  LIN {X -5735.893,Y 2029.899,Z -132.531,A -90.03341,B 0.00000,C -180.00000} ; preinsert
  LIN {X -5735.893,Y 2029.899,Z -382.531,A -90.03341,B 0.00000,C -180.00000} ; insert
  LIN {X -5735.893,Y 2029.899,Z -382.531,A -90.03341,B 0.00000,C -180.00000} ; release
  LIN {X -5735.893,Y 2029.899,Z -82.531,A -90.03341,B 0.00000,C -180.00000} ; retreat
  ; Step 3130, bar 1650
  LIN {X -5860.893,Y 2029.899,Z 855.478,A -90.03341,B 0.00000,C -180.00000} ; outside
  LIN {X -5860.893,Y 2029.899,Z -132.531,A -90.03341,B 0.00000,C -180.00000} ; preinsert
  LIN {X -5860.893,Y 2029.899,Z -382.531,A -90.03341,B 0.00000,C -180.00000} ; insert
  LIN {X -5860.893,Y 2029.899,Z -382.531,A -90.03341,B 0.00000,C -180.00000} ; release
  LIN {X -5860.893,Y 2029.899,Z -82.531,A -90.03341,B 0.00000,C -180.00000} ; retreat
  ; Step 3131, bar 1652
  LIN {X -6110.893,Y 2029.899,Z 855.478,A -90.03341,B 0.00000,C -180.00000} ; outside
  LIN {X -6110.893,Y 2029.899,Z -132.531,A -90.03341,B 0.00000,C -180.00000} ; preinsert
  LIN {X -6110.893,Y 2029.899,Z -382.531,A -90.03341,B 0.00000,C -180.00000} ; insert
  LIN {X -6110.893,Y 2029.899,Z -382.531,A -90.03341,B 0.00000,C -180.00000} ; release
  LIN {X -6110.893,Y 2029.899,Z -82.531,A -90.03341,B 0.00000,C -180.00000} ; retreat
  ; Step 3132, bar 1654
  LIN {X -6235.893,Y 2029.899,Z 855.478,A -90.03341,B 0.00000,C -180.00000} ; outside
  LIN {X -6235.893,Y 2029.899,Z -132.531,A -90.03341,B 0.00000,C -180.00000} ; preinsert
  LIN {X -6235.893,Y 2029.899,Z -382.531,A -90.03341,B 0.00000,C -180.00000} ; insert
  LIN {X -6235.893,Y 2029.899,Z -382.531,A -90.03341,B 0.00000,C -180.00000} ; release
  LIN {X -6235.893,Y 2029.899,Z -82.531,A -90.03341,B 0.00000,C -180.00000} ; retreat
  ; Step 3133, bar 1656
  LIN {X -6360.893,Y 2029.899,Z 855.478,A -90.03341,B 0.00000,C -180.00000} ; outside
  LIN {X -6360.893,Y 2029.899,Z -132.531,A -90.03341,B 0.00000,C -180.00000} ; preinsert
  LIN {X -6360.893,Y 2029.899,Z -382.531,A -90.03341,B 0.00000,C -180.00000} ; insert
  LIN {X -6360.893,Y 2029.899,Z -382.531,A -90.03341,B 0.00000,C -180.00000} ; release
  LIN {X -6360.893,Y 2029.899,Z -82.531,A -90.03341,B 0.00000,C -180.00000} ; retreat
  ; Step 3134, bar 1658
  LIN {X -6485.893,Y 2029.899,Z 855.478,A -90.03341,B 0.00000,C -180.00000} ; outside
  LIN {X -6485.893,Y 2029.899,Z -132.531,A -90.03341,B 0.00000,C -180.00000} ; preinsert
  LIN {X -6485.893,Y 2029.899,Z -382.531,A -90.03341,B 0.00000,C -180.00000} ; insert
  LIN {X -6485.893,Y 2029.899,Z -382.531,A -90.03341,B 0.00000,C -180.00000} ; release
  LIN {X -6485.893,Y 2029.899,Z -82.531,A -90.03341,B 0.00000,C -180.00000} ; retreat
  ; Step 3135, bar 1660
  LIN {X -6610.893,Y 2029.899,Z 855.478,A -90.03341,B 0.00000,C -180.00000} ; outside
  LIN {X -6610.893,Y 2029.899,Z -132.531,A -90.03341,B 0.00000,C -180.00000} ; preinsert
  LIN {X -6610.893,Y 2029.899,Z -382.531,A -90.03341,B 0.00000,C -180.00000} ; insert
  LIN {X -6610.893,Y 2029.899,Z -382.531,A -90.03341,B 0.00000,C -180.00000} ; release
  LIN {X -6610.893,Y 2029.899,Z -82.531,A -90.03341,B 0.00000,C -180.00000} ; retreat
  ; Step 3136, bar 1662
  LIN {X -6735.893,Y 2029.899,Z 855.478,A -90.03341,B 0.00000,C -180.00000} ; outside
  LIN {X -6735.893,Y 2029.899,Z -132.531,A -90.03341,B 0.00000,C -180.00000} ; preinsert
  LIN {X -6735.893,Y 2029.899,Z -382.531,A -90.03341,B 0.00000,C -180.00000} ; insert
  LIN {X -6735.893,Y 2029.899,Z -382.531,A -90.03341,B 0.00000,C -180.00000} ; release
  LIN {X -6735.893,Y 2029.899,Z -82.531,A -90.03341,B 0.00000,C -180.00000} ; retreat
  ; Step 3137, bar 1664
  LIN {X -6860.893,Y 2029.899,Z 855.478,A -90.03341,B 0.00000,C -180.00000} ; outside
  LIN {X -6860.893,Y 2029.899,Z -132.531,A -90.03341,B 0.00000,C -180.00000} ; preinsert
  LIN {X -6860.893,Y 2029.899,Z -382.531,A -90.03341,B 0.00000,C -180.00000} ; insert
  LIN {X -6860.893,Y 2029.899,Z -382.531,A -90.03341,B 0.00000,C -180.00000} ; release
  LIN {X -6860.893,Y 2029.899,Z -82.531,A -90.03341,B 0.00000,C -180.00000} ; retreat
  ; Step 3138, bar 1666
  LIN {X -6985.893,Y 2029.899,Z 855.478,A -90.03341,B 0.00000,C -180.00000} ; outside
  LIN {X -6985.893,Y 2029.899,Z -132.531,A -90.03341,B 0.00000,C -180.00000} ; preinsert
  LIN {X -6985.893,Y 2029.899,Z -382.531,A -90.03341,B 0.00000,C -180.00000} ; insert
  LIN {X -6985.893,Y 2029.899,Z -382.531,A -90.03341,B 0.00000,C -180.00000} ; release
  LIN {X -6985.893,Y 2029.899,Z -82.531,A -90.03341,B 0.00000,C -180.00000} ; retreat
  ; Step 3139, bar 1668
  LIN {X -7110.893,Y 2029.899,Z 855.478,A -90.03341,B 0.00000,C -180.00000} ; outside
  LIN {X -7110.893,Y 2029.899,Z -132.531,A -90.03341,B 0.00000,C -180.00000} ; preinsert
  LIN {X -7110.893,Y 2029.899,Z -382.531,A -90.03341,B 0.00000,C -180.00000} ; insert
  LIN {X -7110.893,Y 2029.899,Z -382.531,A -90.03341,B 0.00000,C -180.00000} ; release
  LIN {X -7110.893,Y 2029.899,Z -82.531,A -90.03341,B 0.00000,C -180.00000} ; retreat
  ; Step 3140, bar 1670
  LIN {X -7235.893,Y 2029.899,Z 855.478,A -90.03341,B 0.00000,C -180.00000} ; outside
  LIN {X -7235.893,Y 2029.899,Z -132.531,A -90.03341,B 0.00000,C -180.00000} ; preinsert
  LIN {X -7235.893,Y 2029.899,Z -382.531,A -90.03341,B 0.00000,C -180.00000} ; insert
  LIN {X -7235.893,Y 2029.899,Z -382.531,A -90.03341,B 0.00000,C -180.00000} ; release
  LIN {X -7235.893,Y 2029.899,Z -82.531,A -90.03341,B 0.00000,C -180.00000} ; retreat
  ; Step 3141, bar 1672
  LIN {X -7360.893,Y 2029.899,Z 855.478,A -90.03341,B 0.00000,C -180.00000} ; outside
  LIN {X -7360.893,Y 2029.899,Z -132.531,A -90.03341,B 0.00000,C -180.00000} ; preinsert
  LIN {X -7360.893,Y 2029.899,Z -382.531,A -90.03341,B 0.00000,C -180.00000} ; insert
  LIN {X -7360.893,Y 2029.899,Z -382.531,A -90.03341,B 0.00000,C -180.00000} ; release
  LIN {X -7360.893,Y 2029.899,Z -82.531,A -90.03341,B 0.00000,C -180.00000} ; retreat
  ; Step 3142, bar 1674
  LIN {X -7485.893,Y 2029.899,Z 855.478,A -90.03341,B 0.00000,C -180.00000} ; outside
  LIN {X -7485.893,Y 2029.899,Z -132.531,A -90.03341,B 0.00000,C -180.00000} ; preinsert
  LIN {X -7485.893,Y 2029.899,Z -382.531,A -90.03341,B 0.00000,C -180.00000} ; insert
  LIN {X -7485.893,Y 2029.899,Z -382.531,A -90.03341,B 0.00000,C -180.00000} ; release
  LIN {X -7485.893,Y 2029.899,Z -82.531,A -90.03341,B 0.00000,C -180.00000} ; retreat
  ; Step 3143, bar 1676
  LIN {X -7610.893,Y 2029.899,Z 855.478,A -90.03341,B 0.00000,C -180.00000} ; outside
  LIN {X -7610.893,Y 2029.899,Z -132.531,A -90.03341,B 0.00000,C -180.00000} ; preinsert
  LIN {X -7610.893,Y 2029.899,Z -382.531,A -90.03341,B 0.00000,C -180.00000} ; insert
  LIN {X -7610.893,Y 2029.899,Z -382.531,A -90.03341,B 0.00000,C -180.00000} ; release
  LIN {X -7610.893,Y 2029.899,Z -82.531,A -90.03341,B 0.00000,C -180.00000} ; retreat
  ; Step 3144, bar 1678
  LIN {X -7735.893,Y 2029.899,Z 855.478,A -90.03341,B 0.00000,C -180.00000} ; outside
  LIN {X -7735.893,Y 2029.899,Z -132.531,A -90.03341,B 0.00000,C -180.00000} ; preinsert
  LIN {X -7735.893,Y 2029.899,Z -382.531,A -90.03341,B 0.00000,C -180.00000} ; insert
  LIN {X -7735.893,Y 2029.899,Z -382.531,A -90.03341,B 0.00000,C -180.00000} ; release
  LIN {X -7735.893,Y 2029.899,Z -82.531,A -90.03341,B 0.00000,C -180.00000} ; retreat
  ; Step 3145, bar 1680
  LIN {X -7860.893,Y 2029.899,Z 855.478,A -90.03341,B 0.00000,C -180.00000} ; outside
  LIN {X -7860.893,Y 2029.899,Z -132.531,A -90.03341,B 0.00000,C -180.00000} ; preinsert
  LIN {X -7860.893,Y 2029.899,Z -382.531,A -90.03341,B 0.00000,C -180.00000} ; insert
  LIN {X -7860.893,Y 2029.899,Z -382.531,A -90.03341,B 0.00000,C -180.00000} ; release
  LIN {X -7860.893,Y 2029.899,Z -82.531,A -90.03341,B 0.00000,C -180.00000} ; retreat
  ; Step 3146, bar 1682
  LIN {X -7985.893,Y 2029.899,Z 855.478,A -90.03341,B 0.00000,C -180.00000} ; outside
  LIN {X -7985.893,Y 2029.899,Z -132.531,A -90.03341,B 0.00000,C -180.00000} ; preinsert
  LIN {X -7985.893,Y 2029.899,Z -382.531,A -90.03341,B 0.00000,C -180.00000} ; insert
  LIN {X -7985.893,Y 2029.899,Z -382.531,A -90.03341,B 0.00000,C -180.00000} ; release
  LIN {X -7985.893,Y 2029.899,Z -82.531,A -90.03341,B 0.00000,C -180.00000} ; retreat
  ; Step 3147, bar 1684
  LIN {X -8110.893,Y 2029.899,Z 855.478,A -90.03341,B 0.00000,C -180.00000} ; outside
  LIN {X -8110.893,Y 2029.899,Z -132.531,A -90.03341,B 0.00000,C -180.00000} ; preinsert
  LIN {X -8110.893,Y 2029.899,Z -382.531,A -90.03341,B 0.00000,C -180.00000} ; insert
  LIN {X -8110.893,Y 2029.899,Z -382.531,A -90.03341,B 0.00000,C -180.00000} ; release
  LIN {X -8110.893,Y 2029.899,Z -82.531,A -90.03341,B 0.00000,C -180.00000} ; retreat
  ; Step 3148, bar 1686
  LIN {X -8235.893,Y 2029.899,Z 855.478,A -90.03341,B 0.00000,C 180.00000} ; outside
  LIN {X -8235.893,Y 2029.899,Z -132.531,A -90.03341,B 0.00000,C 180.00000} ; preinsert
  LIN {X -8235.893,Y 2029.899,Z -382.531,A -90.03341,B 0.00000,C 180.00000} ; insert
  LIN {X -8235.893,Y 2029.899,Z -382.531,A -90.03341,B 0.00000,C 180.00000} ; release
  LIN {X -8235.893,Y 2029.899,Z -82.531,A -90.03341,B 0.00000,C 180.00000} ; retreat
  ; Step 3149, bar 1688
  LIN {X -8360.893,Y 2029.899,Z 855.478,A -90.03341,B 0.00000,C 180.00000} ; outside
  LIN {X -8360.893,Y 2029.899,Z -132.531,A -90.03341,B 0.00000,C 180.00000} ; preinsert
  LIN {X -8360.893,Y 2029.899,Z -382.531,A -90.03341,B 0.00000,C 180.00000} ; insert
  LIN {X -8360.893,Y 2029.899,Z -382.531,A -90.03341,B 0.00000,C 180.00000} ; release
  LIN {X -8360.893,Y 2029.899,Z -82.531,A -90.03341,B 0.00000,C 180.00000} ; retreat
  ; Step 3150, bar 1690
  LIN {X -8485.893,Y 2029.899,Z 855.478,A -90.03341,B 0.00000,C 180.00000} ; outside
  LIN {X -8485.893,Y 2029.899,Z -132.531,A -90.03341,B 0.00000,C 180.00000} ; preinsert
  LIN {X -8485.893,Y 2029.899,Z -382.531,A -90.03341,B 0.00000,C 180.00000} ; insert
  LIN {X -8485.893,Y 2029.899,Z -382.531,A -90.03341,B 0.00000,C 180.00000} ; release
  LIN {X -8485.893,Y 2029.899,Z -82.531,A -90.03341,B 0.00000,C 180.00000} ; retreat
  ; Step 3151, bar 1692
  LIN {X -8610.893,Y 2029.899,Z 855.478,A -90.03341,B 0.00000,C 180.00000} ; outside
  LIN {X -8610.893,Y 2029.899,Z -132.531,A -90.03341,B 0.00000,C 180.00000} ; preinsert
  LIN {X -8610.893,Y 2029.899,Z -382.531,A -90.03341,B 0.00000,C 180.00000} ; insert
  LIN {X -8610.893,Y 2029.899,Z -382.531,A -90.03341,B 0.00000,C 180.00000} ; release
  LIN {X -8610.893,Y 2029.899,Z -82.531,A -90.03341,B 0.00000,C 180.00000} ; retreat
  ; Step 3152, bar 1694
  LIN {X -8735.893,Y 2029.899,Z 855.478,A -90.03341,B 0.00000,C 180.00000} ; outside
  LIN {X -8735.893,Y 2029.899,Z -132.531,A -90.03341,B 0.00000,C 180.00000} ; preinsert
  LIN {X -8735.893,Y 2029.899,Z -382.531,A -90.03341,B 0.00000,C 180.00000} ; insert
  LIN {X -8735.893,Y 2029.899,Z -382.531,A -90.03341,B 0.00000,C 180.00000} ; release
  LIN {X -8735.893,Y 2029.899,Z -82.531,A -90.03341,B 0.00000,C 180.00000} ; retreat
  ; Step 3153, bar 1696
  LIN {X -8860.893,Y 2029.899,Z 855.478,A -90.03341,B 0.00000,C 180.00000} ; outside
  LIN {X -8860.893,Y 2029.899,Z -132.531,A -90.03341,B 0.00000,C 180.00000} ; preinsert
  LIN {X -8860.893,Y 2029.899,Z -382.531,A -90.03341,B 0.00000,C 180.00000} ; insert
  LIN {X -8860.893,Y 2029.899,Z -382.531,A -90.03341,B 0.00000,C 180.00000} ; release
  LIN {X -8860.893,Y 2029.899,Z -82.531,A -90.03341,B 0.00000,C 180.00000} ; retreat
  ; Step 3154, bar 1698
  LIN {X -8985.893,Y 2029.899,Z 855.478,A -90.03341,B 0.00000,C 180.00000} ; outside
  LIN {X -8985.893,Y 2029.899,Z -132.531,A -90.03341,B 0.00000,C 180.00000} ; preinsert
  LIN {X -8985.893,Y 2029.899,Z -382.531,A -90.03341,B 0.00000,C 180.00000} ; insert
  LIN {X -8985.893,Y 2029.899,Z -382.531,A -90.03341,B 0.00000,C 180.00000} ; release
  LIN {X -8985.893,Y 2029.899,Z -82.531,A -90.03341,B 0.00000,C 180.00000} ; retreat
  ; Step 3155, bar 1700
  LIN {X -9110.893,Y 2029.899,Z 855.478,A -90.03341,B 0.00000,C 180.00000} ; outside
  LIN {X -9110.893,Y 2029.899,Z -132.531,A -90.03341,B 0.00000,C 180.00000} ; preinsert
  LIN {X -9110.893,Y 2029.899,Z -382.531,A -90.03341,B 0.00000,C 180.00000} ; insert
  LIN {X -9110.893,Y 2029.899,Z -382.531,A -90.03341,B 0.00000,C 180.00000} ; release
  LIN {X -9110.893,Y 2029.899,Z -82.531,A -90.03341,B 0.00000,C 180.00000} ; retreat
  ; Step 3156, bar 1702
  LIN {X -9235.893,Y 2029.899,Z 855.478,A -90.03341,B 0.00000,C 180.00000} ; outside
  LIN {X -9235.893,Y 2029.899,Z -132.531,A -90.03341,B 0.00000,C 180.00000} ; preinsert
  LIN {X -9235.893,Y 2029.899,Z -382.531,A -90.03341,B 0.00000,C 180.00000} ; insert
  LIN {X -9235.893,Y 2029.899,Z -382.531,A -90.03341,B 0.00000,C 180.00000} ; release
  LIN {X -9235.893,Y 2029.899,Z -82.531,A -90.03341,B 0.00000,C 180.00000} ; retreat
  ; Step 3157, bar 1704
  LIN {X -9360.893,Y 2029.899,Z 855.478,A -90.03341,B 0.00000,C 180.00000} ; outside
  LIN {X -9360.893,Y 2029.899,Z -132.531,A -90.03341,B 0.00000,C 180.00000} ; preinsert
  LIN {X -9360.893,Y 2029.899,Z -382.531,A -90.03341,B 0.00000,C 180.00000} ; insert
  LIN {X -9360.893,Y 2029.899,Z -382.531,A -90.03341,B 0.00000,C 180.00000} ; release
  LIN {X -9360.893,Y 2029.899,Z -82.531,A -90.03341,B 0.00000,C 180.00000} ; retreat
  ; Step 3158, bar 1706
  LIN {X -9485.893,Y 2029.899,Z 855.478,A -90.03341,B 0.00000,C 180.00000} ; outside
  LIN {X -9485.893,Y 2029.899,Z -132.531,A -90.03341,B 0.00000,C 180.00000} ; preinsert
  LIN {X -9485.893,Y 2029.899,Z -382.531,A -90.03341,B 0.00000,C 180.00000} ; insert
  LIN {X -9485.893,Y 2029.899,Z -382.531,A -90.03341,B 0.00000,C 180.00000} ; release
  LIN {X -9485.893,Y 2029.899,Z -82.531,A -90.03341,B 0.00000,C 180.00000} ; retreat
  ; Step 3159, bar 1708
  LIN {X -9610.893,Y 2029.899,Z 855.478,A -90.03341,B 0.00000,C 180.00000} ; outside
  LIN {X -9610.893,Y 2029.899,Z -132.531,A -90.03341,B 0.00000,C 180.00000} ; preinsert
  LIN {X -9610.893,Y 2029.899,Z -382.531,A -90.03341,B 0.00000,C 180.00000} ; insert
  LIN {X -9610.893,Y 2029.899,Z -382.531,A -90.03341,B 0.00000,C 180.00000} ; release
  LIN {X -9610.893,Y 2029.899,Z -82.531,A -90.03341,B 0.00000,C 180.00000} ; retreat
  ; Step 3160, bar 1710
  LIN {X -9735.893,Y 2029.899,Z 855.478,A -90.03341,B 0.00000,C 180.00000} ; outside
  LIN {X -9735.893,Y 2029.899,Z -132.531,A -90.03341,B 0.00000,C 180.00000} ; preinsert
  LIN {X -9735.893,Y 2029.899,Z -382.531,A -90.03341,B 0.00000,C 180.00000} ; insert
  LIN {X -9735.893,Y 2029.899,Z -382.531,A -90.03341,B 0.00000,C 180.00000} ; release
  LIN {X -9735.893,Y 2029.899,Z -82.531,A -90.03341,B 0.00000,C 180.00000} ; retreat
  ; Step 3161, bar 1712
  LIN {X -9860.893,Y 2029.899,Z 855.478,A -90.03341,B 0.00000,C 180.00000} ; outside
  LIN {X -9860.893,Y 2029.899,Z -132.531,A -90.03341,B 0.00000,C 180.00000} ; preinsert
  LIN {X -9860.893,Y 2029.899,Z -382.531,A -90.03341,B 0.00000,C 180.00000} ; insert
  LIN {X -9860.893,Y 2029.899,Z -382.531,A -90.03341,B 0.00000,C 180.00000} ; release
  LIN {X -9860.893,Y 2029.899,Z -82.531,A -90.03341,B 0.00000,C 180.00000} ; retreat
  ; Step 3162, bar 1714
  LIN {X -10110.893,Y 2029.899,Z 855.478,A -90.03341,B 0.00000,C 180.00000} ; outside
  LIN {X -10110.893,Y 2029.899,Z -132.531,A -90.03341,B 0.00000,C 180.00000} ; preinsert
  LIN {X -10110.893,Y 2029.899,Z -382.531,A -90.03341,B 0.00000,C 180.00000} ; insert
  LIN {X -10110.893,Y 2029.899,Z -382.531,A -90.03341,B 0.00000,C 180.00000} ; release
  LIN {X -10110.893,Y 2029.899,Z -82.531,A -90.03341,B 0.00000,C 180.00000} ; retreat
  ; Step 3163, bar 1716
  LIN {X -10235.893,Y 2029.899,Z 855.478,A -90.03341,B 0.00000,C 180.00000} ; outside
  LIN {X -10235.893,Y 2029.899,Z -132.531,A -90.03341,B 0.00000,C 180.00000} ; preinsert
  LIN {X -10235.893,Y 2029.899,Z -382.531,A -90.03341,B 0.00000,C 180.00000} ; insert
  LIN {X -10235.893,Y 2029.899,Z -382.531,A -90.03341,B 0.00000,C 180.00000} ; release
  LIN {X -10235.893,Y 2029.899,Z -82.531,A -90.03341,B 0.00000,C 180.00000} ; retreat
  ; Step 3164, bar 1718
  LIN {X -10360.893,Y 2029.899,Z 855.478,A -90.03341,B 0.00000,C 180.00000} ; outside
  LIN {X -10360.893,Y 2029.899,Z -132.531,A -90.03341,B 0.00000,C 180.00000} ; preinsert
  LIN {X -10360.893,Y 2029.899,Z -382.531,A -90.03341,B 0.00000,C 180.00000} ; insert
  LIN {X -10360.893,Y 2029.899,Z -382.531,A -90.03341,B 0.00000,C 180.00000} ; release
  LIN {X -10360.893,Y 2029.899,Z -82.531,A -90.03341,B 0.00000,C 180.00000} ; retreat
  ; Step 3165, bar 1720
  LIN {X -10485.893,Y 2029.899,Z 855.478,A -90.03341,B 0.00000,C 180.00000} ; outside
  LIN {X -10485.893,Y 2029.899,Z -132.531,A -90.03341,B 0.00000,C 180.00000} ; preinsert
  LIN {X -10485.893,Y 2029.899,Z -382.531,A -90.03341,B 0.00000,C 180.00000} ; insert
  LIN {X -10485.893,Y 2029.899,Z -382.531,A -90.03341,B 0.00000,C 180.00000} ; release
  LIN {X -10485.893,Y 2029.899,Z -82.531,A -90.03341,B 0.00000,C 180.00000} ; retreat
  ; Step 3166, bar 1722
  LIN {X -10610.893,Y 2029.899,Z 855.478,A -90.03341,B 0.00000,C 180.00000} ; outside
  LIN {X -10610.893,Y 2029.899,Z -132.531,A -90.03341,B 0.00000,C 180.00000} ; preinsert
  LIN {X -10610.893,Y 2029.899,Z -382.531,A -90.03341,B 0.00000,C 180.00000} ; insert
  LIN {X -10610.893,Y 2029.899,Z -382.531,A -90.03341,B 0.00000,C 180.00000} ; release
  LIN {X -10610.893,Y 2029.899,Z -82.531,A -90.03341,B 0.00000,C 180.00000} ; retreat
  ; Step 3167, bar 1724
  LIN {X -10735.893,Y 2029.899,Z 855.478,A -90.03341,B 0.00000,C 180.00000} ; outside
  LIN {X -10735.893,Y 2029.899,Z -132.531,A -90.03341,B 0.00000,C 180.00000} ; preinsert
  LIN {X -10735.893,Y 2029.899,Z -382.531,A -90.03341,B 0.00000,C 180.00000} ; insert
  LIN {X -10735.893,Y 2029.899,Z -382.531,A -90.03341,B 0.00000,C 180.00000} ; release
  LIN {X -10735.893,Y 2029.899,Z -82.531,A -90.03341,B 0.00000,C 180.00000} ; retreat
  ; Step 3168, bar 1726
  LIN {X -10860.893,Y 2029.899,Z 855.478,A -90.03341,B 0.00000,C 180.00000} ; outside
  LIN {X -10860.893,Y 2029.899,Z -132.531,A -90.03341,B 0.00000,C 180.00000} ; preinsert
  LIN {X -10860.893,Y 2029.899,Z -382.531,A -90.03341,B 0.00000,C 180.00000} ; insert
  LIN {X -10860.893,Y 2029.899,Z -382.531,A -90.03341,B 0.00000,C 180.00000} ; release
  LIN {X -10860.893,Y 2029.899,Z -82.531,A -90.03341,B 0.00000,C 180.00000} ; retreat
  ; Step 3169, bar 1728
  LIN {X -10985.893,Y 2029.899,Z 855.478,A -90.03341,B 0.00000,C 180.00000} ; outside
  LIN {X -10985.893,Y 2029.899,Z -132.531,A -90.03341,B 0.00000,C 180.00000} ; preinsert
  LIN {X -10985.893,Y 2029.899,Z -382.531,A -90.03341,B 0.00000,C 180.00000} ; insert
  LIN {X -10985.893,Y 2029.899,Z -382.531,A -90.03341,B 0.00000,C 180.00000} ; release
  LIN {X -10985.893,Y 2029.899,Z -82.531,A -90.03341,B 0.00000,C 180.00000} ; retreat
  ; Step 3170, bar 1730
  LIN {X -11110.893,Y 2029.899,Z 855.478,A -90.03341,B 0.00000,C 180.00000} ; outside
  LIN {X -11110.893,Y 2029.899,Z -132.531,A -90.03341,B 0.00000,C 180.00000} ; preinsert
  LIN {X -11110.893,Y 2029.899,Z -382.531,A -90.03341,B 0.00000,C 180.00000} ; insert
  LIN {X -11110.893,Y 2029.899,Z -382.531,A -90.03341,B 0.00000,C 180.00000} ; release
  LIN {X -11110.893,Y 2029.899,Z -82.531,A -90.03341,B 0.00000,C 180.00000} ; retreat
  ; Step 3171, bar 1732
  LIN {X -11235.893,Y 2029.899,Z 855.478,A -90.03341,B 0.00000,C 180.00000} ; outside
  LIN {X -11235.893,Y 2029.899,Z -132.531,A -90.03341,B 0.00000,C 180.00000} ; preinsert
  LIN {X -11235.893,Y 2029.899,Z -382.531,A -90.03341,B 0.00000,C 180.00000} ; insert
  LIN {X -11235.893,Y 2029.899,Z -382.531,A -90.03341,B 0.00000,C 180.00000} ; release
  LIN {X -11235.893,Y 2029.899,Z -82.531,A -90.03341,B 0.00000,C 180.00000} ; retreat
  ; Step 3172, bar 1734
  LIN {X -11360.893,Y 2029.899,Z 855.478,A -90.03341,B 0.00000,C 180.00000} ; outside
  LIN {X -11360.893,Y 2029.899,Z -132.531,A -90.03341,B 0.00000,C 180.00000} ; preinsert
  LIN {X -11360.893,Y 2029.899,Z -382.531,A -90.03341,B 0.00000,C 180.00000} ; insert
  LIN {X -11360.893,Y 2029.899,Z -382.531,A -90.03341,B 0.00000,C 180.00000} ; release
  LIN {X -11360.893,Y 2029.899,Z -82.531,A -90.03341,B 0.00000,C 180.00000} ; retreat
  ; Step 3173, bar 1736
  LIN {X -11485.893,Y 2029.899,Z 855.478,A -90.03341,B 0.00000,C 180.00000} ; outside
  LIN {X -11485.893,Y 2029.899,Z -132.531,A -90.03341,B 0.00000,C 180.00000} ; preinsert
  LIN {X -11485.893,Y 2029.899,Z -382.531,A -90.03341,B 0.00000,C 180.00000} ; insert
  LIN {X -11485.893,Y 2029.899,Z -382.531,A -90.03341,B 0.00000,C 180.00000} ; release
  LIN {X -11485.893,Y 2029.899,Z -82.531,A -90.03341,B 0.00000,C 180.00000} ; retreat
  ; Step 3174, bar 1738
  LIN {X -11610.893,Y 2029.899,Z 855.478,A -90.03341,B 0.00000,C 180.00000} ; outside
  LIN {X -11610.893,Y 2029.899,Z -132.531,A -90.03341,B 0.00000,C 180.00000} ; preinsert
  LIN {X -11610.893,Y 2029.899,Z -382.531,A -90.03341,B 0.00000,C 180.00000} ; insert
  LIN {X -11610.893,Y 2029.899,Z -382.531,A -90.03341,B 0.00000,C 180.00000} ; release
  LIN {X -11610.893,Y 2029.899,Z -82.531,A -90.03341,B 0.00000,C 180.00000} ; retreat
  ; Step 3175, bar 1740
  LIN {X -11735.893,Y 2029.899,Z 855.478,A -90.03341,B 0.00000,C 180.00000} ; outside
  LIN {X -11735.893,Y 2029.899,Z -132.531,A -90.03341,B 0.00000,C 180.00000} ; preinsert
  LIN {X -11735.893,Y 2029.899,Z -382.531,A -90.03341,B 0.00000,C 180.00000} ; insert
  LIN {X -11735.893,Y 2029.899,Z -382.531,A -90.03341,B 0.00000,C 180.00000} ; release
  LIN {X -11735.893,Y 2029.899,Z -82.531,A -90.03341,B 0.00000,C 180.00000} ; retreat
  ; Step 3176, bar 1742
  LIN {X -11860.893,Y 2029.899,Z 855.478,A -90.03341,B 0.00000,C 180.00000} ; outside
  LIN {X -11860.893,Y 2029.899,Z -132.531,A -90.03341,B 0.00000,C 180.00000} ; preinsert
  LIN {X -11860.893,Y 2029.899,Z -382.531,A -90.03341,B 0.00000,C 180.00000} ; insert
  LIN {X -11860.893,Y 2029.899,Z -382.531,A -90.03341,B 0.00000,C 180.00000} ; release
  LIN {X -11860.893,Y 2029.899,Z -82.531,A -90.03341,B 0.00000,C 180.00000} ; retreat
  ; Step 3177, bar 1744
  LIN {X -11985.893,Y 2029.899,Z 855.478,A -90.03341,B 0.00000,C 180.00000} ; outside
  LIN {X -11985.893,Y 2029.899,Z -132.531,A -90.03341,B 0.00000,C 180.00000} ; preinsert
  LIN {X -11985.893,Y 2029.899,Z -382.531,A -90.03341,B 0.00000,C 180.00000} ; insert
  LIN {X -11985.893,Y 2029.899,Z -382.531,A -90.03341,B 0.00000,C 180.00000} ; release
  LIN {X -11985.893,Y 2029.899,Z -82.531,A -90.03341,B 0.00000,C 180.00000} ; retreat
  ; Step 3178, bar 1746
  LIN {X -12110.893,Y 2029.899,Z 855.478,A -90.03341,B 0.00000,C 180.00000} ; outside
  LIN {X -12110.893,Y 2029.899,Z -132.531,A -90.03341,B 0.00000,C 180.00000} ; preinsert
  LIN {X -12110.893,Y 2029.899,Z -382.531,A -90.03341,B 0.00000,C 180.00000} ; insert
  LIN {X -12110.893,Y 2029.899,Z -382.531,A -90.03341,B 0.00000,C 180.00000} ; release
  LIN {X -12110.893,Y 2029.899,Z -82.531,A -90.03341,B 0.00000,C 180.00000} ; retreat
  ; Step 3179, bar 1748
  LIN {X -12235.893,Y 2029.899,Z 855.478,A -90.03341,B 0.00000,C 180.00000} ; outside
  LIN {X -12235.893,Y 2029.899,Z -132.531,A -90.03341,B 0.00000,C 180.00000} ; preinsert
  LIN {X -12235.893,Y 2029.899,Z -382.531,A -90.03341,B 0.00000,C 180.00000} ; insert
  LIN {X -12235.893,Y 2029.899,Z -382.531,A -90.03341,B 0.00000,C 180.00000} ; release
  LIN {X -12235.893,Y 2029.899,Z -82.531,A -90.03341,B 0.00000,C 180.00000} ; retreat
  ; Step 3180, bar 1750
  LIN {X -12335.893,Y 2029.899,Z 855.478,A -90.03341,B 0.00000,C 180.00000} ; outside
  LIN {X -12335.893,Y 2029.899,Z -132.531,A -90.03341,B 0.00000,C 180.00000} ; preinsert
  LIN {X -12335.893,Y 2029.899,Z -382.531,A -90.03341,B 0.00000,C 180.00000} ; insert
  LIN {X -12335.893,Y 2029.899,Z -382.531,A -90.03341,B 0.00000,C 180.00000} ; release
  LIN {X -12335.893,Y 2029.899,Z -82.531,A -90.03341,B 0.00000,C 180.00000} ; retreat
  ; Step 3181, bar 1752
  LIN {X -12435.893,Y 2029.899,Z 855.478,A -90.03341,B 0.00000,C 180.00000} ; outside
  LIN {X -12435.893,Y 2029.899,Z -132.531,A -90.03341,B 0.00000,C 180.00000} ; preinsert
  LIN {X -12435.893,Y 2029.899,Z -382.531,A -90.03341,B 0.00000,C 180.00000} ; insert
  LIN {X -12435.893,Y 2029.899,Z -382.531,A -90.03341,B 0.00000,C 180.00000} ; release
  LIN {X -12435.893,Y 2029.899,Z -82.531,A -90.03341,B 0.00000,C 180.00000} ; retreat
  ; Step 3182, bar 1754
  LIN {X -12535.893,Y 2029.899,Z 855.478,A -90.03341,B 0.00000,C 180.00000} ; outside
  LIN {X -12535.893,Y 2029.899,Z -132.531,A -90.03341,B 0.00000,C 180.00000} ; preinsert
  LIN {X -12535.893,Y 2029.899,Z -382.531,A -90.03341,B 0.00000,C 180.00000} ; insert
  LIN {X -12535.893,Y 2029.899,Z -382.531,A -90.03341,B 0.00000,C 180.00000} ; release
  LIN {X -12535.893,Y 2029.899,Z -82.531,A -90.03341,B 0.00000,C 180.00000} ; retreat
  ; Step 3183, bar 1756
  LIN {X -12635.893,Y 2029.899,Z 855.478,A -90.03341,B 0.00000,C 180.00000} ; outside
  LIN {X -12635.893,Y 2029.899,Z -132.531,A -90.03341,B 0.00000,C 180.00000} ; preinsert
  LIN {X -12635.893,Y 2029.899,Z -382.531,A -90.03341,B 0.00000,C 180.00000} ; insert
  LIN {X -12635.893,Y 2029.899,Z -382.531,A -90.03341,B 0.00000,C 180.00000} ; release
  LIN {X -12635.893,Y 2029.899,Z -82.531,A -90.03341,B 0.00000,C 180.00000} ; retreat
  ; Step 3184, bar 1758
  LIN {X -12735.893,Y 2029.899,Z 855.478,A -90.03341,B 0.00000,C 180.00000} ; outside
  LIN {X -12735.893,Y 2029.899,Z -132.531,A -90.03341,B 0.00000,C 180.00000} ; preinsert
  LIN {X -12735.893,Y 2029.899,Z -382.531,A -90.03341,B 0.00000,C 180.00000} ; insert
  LIN {X -12735.893,Y 2029.899,Z -382.531,A -90.03341,B 0.00000,C 180.00000} ; release
  LIN {X -12735.893,Y 2029.899,Z -82.531,A -90.03341,B 0.00000,C 180.00000} ; retreat
  ; Step 3185, bar 1760
  LIN {X -12835.893,Y 2029.899,Z 855.478,A -90.03341,B 0.00000,C 180.00000} ; outside
  LIN {X -12835.893,Y 2029.899,Z -132.531,A -90.03341,B 0.00000,C 180.00000} ; preinsert
  LIN {X -12835.893,Y 2029.899,Z -382.531,A -90.03341,B 0.00000,C 180.00000} ; insert
  LIN {X -12835.893,Y 2029.899,Z -382.531,A -90.03341,B 0.00000,C 180.00000} ; release
  LIN {X -12835.893,Y 2029.899,Z -82.531,A -90.03341,B 0.00000,C 180.00000} ; retreat
  ; Step 3186, bar 1762
  LIN {X -12935.893,Y 2029.899,Z 855.478,A -90.03341,B 0.00000,C 180.00000} ; outside
  LIN {X -12935.893,Y 2029.899,Z -132.531,A -90.03341,B 0.00000,C 180.00000} ; preinsert
  LIN {X -12935.893,Y 2029.899,Z -382.531,A -90.03341,B 0.00000,C 180.00000} ; insert
  LIN {X -12935.893,Y 2029.899,Z -382.531,A -90.03341,B 0.00000,C 180.00000} ; release
  LIN {X -12935.893,Y 2029.899,Z -82.531,A -90.03341,B 0.00000,C 180.00000} ; retreat
  ; Step 3187, bar 1764
  LIN {X -13035.893,Y 2029.899,Z 855.478,A -90.03341,B 0.00000,C 180.00000} ; outside
  LIN {X -13035.893,Y 2029.899,Z -132.531,A -90.03341,B 0.00000,C 180.00000} ; preinsert
  LIN {X -13035.893,Y 2029.899,Z -382.531,A -90.03341,B 0.00000,C 180.00000} ; insert
  LIN {X -13035.893,Y 2029.899,Z -382.531,A -90.03341,B 0.00000,C 180.00000} ; release
  LIN {X -13035.893,Y 2029.899,Z -82.531,A -90.03341,B 0.00000,C 180.00000} ; retreat
  ; Step 3188, bar 1766
  LIN {X -13135.893,Y 2029.899,Z 855.478,A -90.03341,B 0.00000,C 180.00000} ; outside
  LIN {X -13135.893,Y 2029.899,Z -132.531,A -90.03341,B 0.00000,C 180.00000} ; preinsert
  LIN {X -13135.893,Y 2029.899,Z -382.531,A -90.03341,B 0.00000,C 180.00000} ; insert
  LIN {X -13135.893,Y 2029.899,Z -382.531,A -90.03341,B 0.00000,C 180.00000} ; release
  LIN {X -13135.893,Y 2029.899,Z -82.531,A -90.03341,B 0.00000,C 180.00000} ; retreat
  ; Step 3189, bar 1768
  LIN {X -13235.893,Y 2029.899,Z 855.478,A -90.03341,B 0.00000,C 180.00000} ; outside
  LIN {X -13235.893,Y 2029.899,Z -132.531,A -90.03341,B 0.00000,C 180.00000} ; preinsert
  LIN {X -13235.893,Y 2029.899,Z -382.531,A -90.03341,B 0.00000,C 180.00000} ; insert
  LIN {X -13235.893,Y 2029.899,Z -382.531,A -90.03341,B 0.00000,C 180.00000} ; release
  LIN {X -13235.893,Y 2029.899,Z -82.531,A -90.03341,B 0.00000,C 180.00000} ; retreat
  ; Step 3190, bar 1770
  LIN {X -13335.893,Y 2029.899,Z 855.478,A -90.03341,B 0.00000,C 180.00000} ; outside
  LIN {X -13335.893,Y 2029.899,Z -132.531,A -90.03341,B 0.00000,C 180.00000} ; preinsert
  LIN {X -13335.893,Y 2029.899,Z -382.531,A -90.03341,B 0.00000,C 180.00000} ; insert
  LIN {X -13335.893,Y 2029.899,Z -382.531,A -90.03341,B 0.00000,C 180.00000} ; release
  LIN {X -13335.893,Y 2029.899,Z -82.531,A -90.03341,B 0.00000,C 180.00000} ; retreat
  ; Step 3191, bar 1774
  LIN {X -13535.893,Y 2029.899,Z 855.478,A -90.03341,B 0.00000,C 180.00000} ; outside
  LIN {X -13535.893,Y 2029.899,Z -132.531,A -90.03341,B 0.00000,C 180.00000} ; preinsert
  LIN {X -13535.893,Y 2029.899,Z -382.531,A -90.03341,B 0.00000,C 180.00000} ; insert
  LIN {X -13535.893,Y 2029.899,Z -382.531,A -90.03341,B 0.00000,C 180.00000} ; release
  LIN {X -13535.893,Y 2029.899,Z -82.531,A -90.03341,B 0.00000,C 180.00000} ; retreat
  ; Step 3192, bar 1772
  LIN {X -13435.893,Y 2029.899,Z 855.478,A -90.03341,B 0.00000,C 180.00000} ; outside
  LIN {X -13435.893,Y 2029.899,Z -132.531,A -90.03341,B 0.00000,C 180.00000} ; preinsert
  LIN {X -13435.893,Y 2029.899,Z -382.531,A -90.03341,B 0.00000,C 180.00000} ; insert
  LIN {X -13435.893,Y 2029.899,Z -382.531,A -90.03341,B 0.00000,C 180.00000} ; release
  LIN {X -13435.893,Y 2029.899,Z -82.531,A -90.03341,B 0.00000,C 180.00000} ; retreat
  ; Step 3193, bar 1776
  LIN {X -13635.893,Y 2029.899,Z 855.478,A -90.03341,B 0.00000,C 180.00000} ; outside
  LIN {X -13635.893,Y 2029.899,Z -132.531,A -90.03341,B 0.00000,C 180.00000} ; preinsert
  LIN {X -13635.893,Y 2029.899,Z -382.531,A -90.03341,B 0.00000,C 180.00000} ; insert
  LIN {X -13635.893,Y 2029.899,Z -382.531,A -90.03341,B 0.00000,C 180.00000} ; release
  LIN {X -13635.893,Y 2029.899,Z -82.531,A -90.03341,B 0.00000,C 180.00000} ; retreat
  ; Step 3194, bar 1778
  LIN {X -13735.893,Y 2029.899,Z 855.478,A -90.03341,B 0.00000,C 180.00000} ; outside
  LIN {X -13735.893,Y 2029.899,Z -132.531,A -90.03341,B 0.00000,C 180.00000} ; preinsert
  LIN {X -13735.893,Y 2029.899,Z -382.531,A -90.03341,B 0.00000,C 180.00000} ; insert
  LIN {X -13735.893,Y 2029.899,Z -382.531,A -90.03341,B 0.00000,C 180.00000} ; release
  LIN {X -13735.893,Y 2029.899,Z -82.531,A -90.03341,B 0.00000,C 180.00000} ; retreat
  ; Step 3195, bar 1780
  LIN {X -13835.893,Y 2029.899,Z 855.478,A -90.03341,B 0.00000,C 180.00000} ; outside
  LIN {X -13835.893,Y 2029.899,Z -132.531,A -90.03341,B 0.00000,C 180.00000} ; preinsert
  LIN {X -13835.893,Y 2029.899,Z -382.531,A -90.03341,B 0.00000,C 180.00000} ; insert
  LIN {X -13835.893,Y 2029.899,Z -382.531,A -90.03341,B 0.00000,C 180.00000} ; release
  LIN {X -13835.893,Y 2029.899,Z -82.531,A -90.03341,B 0.00000,C 180.00000} ; retreat
  ; Step 3196, bar 1782
  LIN {X -14135.893,Y 2029.899,Z 855.478,A -90.03341,B 0.00000,C 180.00000} ; outside
  LIN {X -14135.893,Y 2029.899,Z -132.531,A -90.03341,B 0.00000,C 180.00000} ; preinsert
  LIN {X -14135.893,Y 2029.899,Z -382.531,A -90.03341,B 0.00000,C 180.00000} ; insert
  LIN {X -14135.893,Y 2029.899,Z -382.531,A -90.03341,B 0.00000,C 180.00000} ; release
  LIN {X -14135.893,Y 2029.899,Z -82.531,A -90.03341,B 0.00000,C 180.00000} ; retreat
  ; Step 3197, bar 1784
  LIN {X -14235.893,Y 2029.899,Z 855.478,A -90.03341,B 0.00000,C 180.00000} ; outside
  LIN {X -14235.893,Y 2029.899,Z -132.531,A -90.03341,B 0.00000,C 180.00000} ; preinsert
  LIN {X -14235.893,Y 2029.899,Z -382.531,A -90.03341,B 0.00000,C 180.00000} ; insert
  LIN {X -14235.893,Y 2029.899,Z -382.531,A -90.03341,B 0.00000,C 180.00000} ; release
  LIN {X -14235.893,Y 2029.899,Z -82.531,A -90.03341,B 0.00000,C 180.00000} ; retreat
  ; Step 3198, bar 1252
  LIN {X -14.107,Y 2029.899,Z 855.478,A -89.96659,B 0.00000,C 180.00000} ; outside
  LIN {X -14.107,Y 2029.899,Z -132.531,A -89.96659,B 0.00000,C 180.00000} ; preinsert
  LIN {X -14.107,Y 2029.899,Z -382.531,A -89.96659,B 0.00000,C 180.00000} ; insert
  LIN {X -14.107,Y 2029.899,Z -382.531,A -89.96659,B 0.00000,C 180.00000} ; release
  LIN {X -14.107,Y 2029.899,Z -82.531,A -89.96659,B 0.00000,C 180.00000} ; retreat
  ; Step 3199, bar 1254
  LIN {X 110.893,Y 2029.899,Z 855.478,A -89.96659,B 0.00000,C 180.00000} ; outside
  LIN {X 110.893,Y 2029.899,Z -132.531,A -89.96659,B 0.00000,C 180.00000} ; preinsert
  LIN {X 110.893,Y 2029.899,Z -382.531,A -89.96659,B 0.00000,C 180.00000} ; insert
  LIN {X 110.893,Y 2029.899,Z -382.531,A -89.96659,B 0.00000,C 180.00000} ; release
  LIN {X 110.893,Y 2029.899,Z -82.531,A -89.96659,B 0.00000,C 180.00000} ; retreat
  ; Step 3200, bar 1256
  LIN {X 235.893,Y 2029.899,Z 855.478,A -89.96659,B 0.00000,C 180.00000} ; outside
  LIN {X 235.893,Y 2029.899,Z -132.531,A -89.96659,B 0.00000,C 180.00000} ; preinsert
  LIN {X 235.893,Y 2029.899,Z -382.531,A -89.96659,B 0.00000,C 180.00000} ; insert
  LIN {X 235.893,Y 2029.899,Z -382.531,A -89.96659,B 0.00000,C 180.00000} ; release
  LIN {X 235.893,Y 2029.899,Z -82.531,A -89.96659,B 0.00000,C 180.00000} ; retreat
  ; Step 3201, bar 1258
  LIN {X 360.893,Y 2029.899,Z 855.478,A -89.96659,B 0.00000,C 180.00000} ; outside
  LIN {X 360.893,Y 2029.899,Z -132.531,A -89.96659,B 0.00000,C 180.00000} ; preinsert
  LIN {X 360.893,Y 2029.899,Z -382.531,A -89.96659,B 0.00000,C 180.00000} ; insert
  LIN {X 360.893,Y 2029.899,Z -382.531,A -89.96659,B 0.00000,C 180.00000} ; release
  LIN {X 360.893,Y 2029.899,Z -82.531,A -89.96659,B 0.00000,C 180.00000} ; retreat
  ; Step 3202, bar 1260
  LIN {X 485.893,Y 2029.899,Z 855.478,A -89.96659,B 0.00000,C 180.00000} ; outside
  LIN {X 485.893,Y 2029.899,Z -132.531,A -89.96659,B 0.00000,C 180.00000} ; preinsert
  LIN {X 485.893,Y 2029.899,Z -382.531,A -89.96659,B 0.00000,C 180.00000} ; insert
  LIN {X 485.893,Y 2029.899,Z -382.531,A -89.96659,B 0.00000,C 180.00000} ; release
  LIN {X 485.893,Y 2029.899,Z -82.531,A -89.96659,B 0.00000,C 180.00000} ; retreat
  ; Step 3203, bar 1262
  LIN {X 610.893,Y 2029.899,Z 855.478,A -89.96659,B 0.00000,C 180.00000} ; outside
  LIN {X 610.893,Y 2029.899,Z -132.531,A -89.96659,B 0.00000,C 180.00000} ; preinsert
  LIN {X 610.893,Y 2029.899,Z -382.531,A -89.96659,B 0.00000,C 180.00000} ; insert
  LIN {X 610.893,Y 2029.899,Z -382.531,A -89.96659,B 0.00000,C 180.00000} ; release
  LIN {X 610.893,Y 2029.899,Z -82.531,A -89.96659,B 0.00000,C 180.00000} ; retreat
  ; Step 3204, bar 1264
  LIN {X 735.893,Y 2029.899,Z 855.478,A -89.96659,B 0.00000,C 180.00000} ; outside
  LIN {X 735.893,Y 2029.899,Z -132.531,A -89.96659,B 0.00000,C 180.00000} ; preinsert
  LIN {X 735.893,Y 2029.899,Z -382.531,A -89.96659,B 0.00000,C 180.00000} ; insert
  LIN {X 735.893,Y 2029.899,Z -382.531,A -89.96659,B 0.00000,C 180.00000} ; release
  LIN {X 735.893,Y 2029.899,Z -82.531,A -89.96659,B 0.00000,C 180.00000} ; retreat
  ; Step 3205, bar 1266
  LIN {X 860.893,Y 2029.899,Z 855.478,A -89.96659,B 0.00000,C 180.00000} ; outside
  LIN {X 860.893,Y 2029.899,Z -132.531,A -89.96659,B 0.00000,C 180.00000} ; preinsert
  LIN {X 860.893,Y 2029.899,Z -382.531,A -89.96659,B 0.00000,C 180.00000} ; insert
  LIN {X 860.893,Y 2029.899,Z -382.531,A -89.96659,B 0.00000,C 180.00000} ; release
  LIN {X 860.893,Y 2029.899,Z -82.531,A -89.96659,B 0.00000,C 180.00000} ; retreat
  ; Step 3206, bar 1268
  LIN {X 985.893,Y 2029.899,Z 855.478,A -89.96659,B 0.00000,C 180.00000} ; outside
  LIN {X 985.893,Y 2029.899,Z -132.531,A -89.96659,B 0.00000,C 180.00000} ; preinsert
  LIN {X 985.893,Y 2029.899,Z -382.531,A -89.96659,B 0.00000,C 180.00000} ; insert
  LIN {X 985.893,Y 2029.899,Z -382.531,A -89.96659,B 0.00000,C 180.00000} ; release
  LIN {X 985.893,Y 2029.899,Z -82.531,A -89.96659,B 0.00000,C 180.00000} ; retreat
  ; Step 3207, bar 1270
  LIN {X 1110.893,Y 2029.899,Z 855.478,A -89.96659,B 0.00000,C 180.00000} ; outside
  LIN {X 1110.893,Y 2029.899,Z -132.531,A -89.96659,B 0.00000,C 180.00000} ; preinsert
  LIN {X 1110.893,Y 2029.899,Z -382.531,A -89.96659,B 0.00000,C 180.00000} ; insert
  LIN {X 1110.893,Y 2029.899,Z -382.531,A -89.96659,B 0.00000,C 180.00000} ; release
  LIN {X 1110.893,Y 2029.899,Z -82.531,A -89.96659,B 0.00000,C 180.00000} ; retreat
  ; Step 3208, bar 1272
  LIN {X 1235.893,Y 2029.899,Z 855.478,A -89.96659,B 0.00000,C 180.00000} ; outside
  LIN {X 1235.893,Y 2029.899,Z -132.531,A -89.96659,B 0.00000,C 180.00000} ; preinsert
  LIN {X 1235.893,Y 2029.899,Z -382.531,A -89.96659,B 0.00000,C 180.00000} ; insert
  LIN {X 1235.893,Y 2029.899,Z -382.531,A -89.96659,B 0.00000,C 180.00000} ; release
  LIN {X 1235.893,Y 2029.899,Z -82.531,A -89.96659,B 0.00000,C 180.00000} ; retreat
  ; Step 3209, bar 1274
  LIN {X 1360.893,Y 2029.899,Z 855.478,A -89.96659,B 0.00000,C 180.00000} ; outside
  LIN {X 1360.893,Y 2029.899,Z -132.531,A -89.96659,B 0.00000,C 180.00000} ; preinsert
  LIN {X 1360.893,Y 2029.899,Z -382.531,A -89.96659,B 0.00000,C 180.00000} ; insert
  LIN {X 1360.893,Y 2029.899,Z -382.531,A -89.96659,B 0.00000,C 180.00000} ; release
  LIN {X 1360.893,Y 2029.899,Z -82.531,A -89.96659,B 0.00000,C 180.00000} ; retreat
  ; Step 3210, bar 1276
  LIN {X 1485.893,Y 2029.899,Z 855.478,A -89.96659,B 0.00000,C 180.00000} ; outside
  LIN {X 1485.893,Y 2029.899,Z -132.531,A -89.96659,B 0.00000,C 180.00000} ; preinsert
  LIN {X 1485.893,Y 2029.899,Z -382.531,A -89.96659,B 0.00000,C 180.00000} ; insert
  LIN {X 1485.893,Y 2029.899,Z -382.531,A -89.96659,B 0.00000,C 180.00000} ; release
  LIN {X 1485.893,Y 2029.899,Z -82.531,A -89.96659,B 0.00000,C 180.00000} ; retreat
  ; Step 3211, bar 1278
  LIN {X 1610.893,Y 2029.899,Z 855.478,A -89.96659,B 0.00000,C 180.00000} ; outside
  LIN {X 1610.893,Y 2029.899,Z -132.531,A -89.96659,B 0.00000,C 180.00000} ; preinsert
  LIN {X 1610.893,Y 2029.899,Z -382.531,A -89.96659,B 0.00000,C 180.00000} ; insert
  LIN {X 1610.893,Y 2029.899,Z -382.531,A -89.96659,B 0.00000,C 180.00000} ; release
  LIN {X 1610.893,Y 2029.899,Z -82.531,A -89.96659,B 0.00000,C 180.00000} ; retreat
  ; Step 3212, bar 1280
  LIN {X 1735.893,Y 2029.899,Z 855.478,A -89.96659,B 0.00000,C 180.00000} ; outside
  LIN {X 1735.893,Y 2029.899,Z -132.531,A -89.96659,B 0.00000,C 180.00000} ; preinsert
  LIN {X 1735.893,Y 2029.899,Z -382.531,A -89.96659,B 0.00000,C 180.00000} ; insert
  LIN {X 1735.893,Y 2029.899,Z -382.531,A -89.96659,B 0.00000,C 180.00000} ; release
  LIN {X 1735.893,Y 2029.899,Z -82.531,A -89.96659,B 0.00000,C 180.00000} ; retreat
  ; Step 3213, bar 1282
  LIN {X 1860.893,Y 2029.899,Z 855.478,A -89.96659,B 0.00000,C 180.00000} ; outside
  LIN {X 1860.893,Y 2029.899,Z -132.531,A -89.96659,B 0.00000,C 180.00000} ; preinsert
  LIN {X 1860.893,Y 2029.899,Z -382.531,A -89.96659,B 0.00000,C 180.00000} ; insert
  LIN {X 1860.893,Y 2029.899,Z -382.531,A -89.96659,B 0.00000,C 180.00000} ; release
  LIN {X 1860.893,Y 2029.899,Z -82.531,A -89.96659,B 0.00000,C 180.00000} ; retreat
  ; Step 3214, bar 1284
  LIN {X 2110.893,Y 2029.899,Z 855.478,A -89.96659,B 0.00000,C 180.00000} ; outside
  LIN {X 2110.893,Y 2029.899,Z -132.531,A -89.96659,B 0.00000,C 180.00000} ; preinsert
  LIN {X 2110.893,Y 2029.899,Z -382.531,A -89.96659,B 0.00000,C 180.00000} ; insert
  LIN {X 2110.893,Y 2029.899,Z -382.531,A -89.96659,B 0.00000,C 180.00000} ; release
  LIN {X 2110.893,Y 2029.899,Z -82.531,A -89.96659,B 0.00000,C 180.00000} ; retreat
  ; Step 3215, bar 1286
  LIN {X 2235.893,Y 2029.899,Z 855.478,A -89.96659,B 0.00000,C 180.00000} ; outside
  LIN {X 2235.893,Y 2029.899,Z -132.531,A -89.96659,B 0.00000,C 180.00000} ; preinsert
  LIN {X 2235.893,Y 2029.899,Z -382.531,A -89.96659,B 0.00000,C 180.00000} ; insert
  LIN {X 2235.893,Y 2029.899,Z -382.531,A -89.96659,B 0.00000,C 180.00000} ; release
  LIN {X 2235.893,Y 2029.899,Z -82.531,A -89.96659,B 0.00000,C 180.00000} ; retreat
  ; Step 3216, bar 1288
  LIN {X 2360.893,Y 2029.899,Z 855.478,A -89.96659,B 0.00000,C 180.00000} ; outside
  LIN {X 2360.893,Y 2029.899,Z -132.531,A -89.96659,B 0.00000,C 180.00000} ; preinsert
  LIN {X 2360.893,Y 2029.899,Z -382.531,A -89.96659,B 0.00000,C 180.00000} ; insert
  LIN {X 2360.893,Y 2029.899,Z -382.531,A -89.96659,B 0.00000,C 180.00000} ; release
  LIN {X 2360.893,Y 2029.899,Z -82.531,A -89.96659,B 0.00000,C 180.00000} ; retreat
  ; Step 3217, bar 1290
  LIN {X 2485.893,Y 2029.899,Z 855.478,A -89.96659,B 0.00000,C 180.00000} ; outside
  LIN {X 2485.893,Y 2029.899,Z -132.531,A -89.96659,B 0.00000,C 180.00000} ; preinsert
  LIN {X 2485.893,Y 2029.899,Z -382.531,A -89.96659,B 0.00000,C 180.00000} ; insert
  LIN {X 2485.893,Y 2029.899,Z -382.531,A -89.96659,B 0.00000,C 180.00000} ; release
  LIN {X 2485.893,Y 2029.899,Z -82.531,A -89.96659,B 0.00000,C 180.00000} ; retreat
  ; Step 3218, bar 1292
  LIN {X 2610.893,Y 2029.899,Z 855.478,A -89.96659,B 0.00000,C 180.00000} ; outside
  LIN {X 2610.893,Y 2029.899,Z -132.531,A -89.96659,B 0.00000,C 180.00000} ; preinsert
  LIN {X 2610.893,Y 2029.899,Z -382.531,A -89.96659,B 0.00000,C 180.00000} ; insert
  LIN {X 2610.893,Y 2029.899,Z -382.531,A -89.96659,B 0.00000,C 180.00000} ; release
  LIN {X 2610.893,Y 2029.899,Z -82.531,A -89.96659,B 0.00000,C 180.00000} ; retreat
  ; Step 3219, bar 1294
  LIN {X 2735.893,Y 2029.899,Z 855.478,A -89.96659,B 0.00000,C 180.00000} ; outside
  LIN {X 2735.893,Y 2029.899,Z -132.531,A -89.96659,B 0.00000,C 180.00000} ; preinsert
  LIN {X 2735.893,Y 2029.899,Z -382.531,A -89.96659,B 0.00000,C 180.00000} ; insert
  LIN {X 2735.893,Y 2029.899,Z -382.531,A -89.96659,B 0.00000,C 180.00000} ; release
  LIN {X 2735.893,Y 2029.899,Z -82.531,A -89.96659,B 0.00000,C 180.00000} ; retreat
  ; Step 3220, bar 1296
  LIN {X 2860.893,Y 2029.899,Z 855.478,A -89.96659,B 0.00000,C 180.00000} ; outside
  LIN {X 2860.893,Y 2029.899,Z -132.531,A -89.96659,B 0.00000,C 180.00000} ; preinsert
  LIN {X 2860.893,Y 2029.899,Z -382.531,A -89.96659,B 0.00000,C 180.00000} ; insert
  LIN {X 2860.893,Y 2029.899,Z -382.531,A -89.96659,B 0.00000,C 180.00000} ; release
  LIN {X 2860.893,Y 2029.899,Z -82.531,A -89.96659,B 0.00000,C 180.00000} ; retreat
  ; Step 3221, bar 1298
  LIN {X 2985.893,Y 2029.899,Z 855.478,A -89.96659,B 0.00000,C 180.00000} ; outside
  LIN {X 2985.893,Y 2029.899,Z -132.531,A -89.96659,B 0.00000,C 180.00000} ; preinsert
  LIN {X 2985.893,Y 2029.899,Z -382.531,A -89.96659,B 0.00000,C 180.00000} ; insert
  LIN {X 2985.893,Y 2029.899,Z -382.531,A -89.96659,B 0.00000,C 180.00000} ; release
  LIN {X 2985.893,Y 2029.899,Z -82.531,A -89.96659,B 0.00000,C 180.00000} ; retreat
  ; Step 3222, bar 1300
  LIN {X 3110.893,Y 2029.899,Z 855.478,A -89.96659,B 0.00000,C 180.00000} ; outside
  LIN {X 3110.893,Y 2029.899,Z -132.531,A -89.96659,B 0.00000,C 180.00000} ; preinsert
  LIN {X 3110.893,Y 2029.899,Z -382.531,A -89.96659,B 0.00000,C 180.00000} ; insert
  LIN {X 3110.893,Y 2029.899,Z -382.531,A -89.96659,B 0.00000,C 180.00000} ; release
  LIN {X 3110.893,Y 2029.899,Z -82.531,A -89.96659,B 0.00000,C 180.00000} ; retreat
  ; Step 3223, bar 1302
  LIN {X 3235.893,Y 2029.899,Z 855.478,A -89.96659,B 0.00000,C 180.00000} ; outside
  LIN {X 3235.893,Y 2029.899,Z -132.531,A -89.96659,B 0.00000,C 180.00000} ; preinsert
  LIN {X 3235.893,Y 2029.899,Z -382.531,A -89.96659,B 0.00000,C 180.00000} ; insert
  LIN {X 3235.893,Y 2029.899,Z -382.531,A -89.96659,B 0.00000,C 180.00000} ; release
  LIN {X 3235.893,Y 2029.899,Z -82.531,A -89.96659,B 0.00000,C 180.00000} ; retreat
  ; Step 3224, bar 1304
  LIN {X 3360.893,Y 2029.899,Z 855.478,A -89.96659,B 0.00000,C 180.00000} ; outside
  LIN {X 3360.893,Y 2029.899,Z -132.531,A -89.96659,B 0.00000,C 180.00000} ; preinsert
  LIN {X 3360.893,Y 2029.899,Z -382.531,A -89.96659,B 0.00000,C 180.00000} ; insert
  LIN {X 3360.893,Y 2029.899,Z -382.531,A -89.96659,B 0.00000,C 180.00000} ; release
  LIN {X 3360.893,Y 2029.899,Z -82.531,A -89.96659,B 0.00000,C 180.00000} ; retreat
  ; Step 3225, bar 1306
  LIN {X 3485.893,Y 2029.899,Z 855.478,A -89.96659,B 0.00000,C 180.00000} ; outside
  LIN {X 3485.893,Y 2029.899,Z -132.531,A -89.96659,B 0.00000,C 180.00000} ; preinsert
  LIN {X 3485.893,Y 2029.899,Z -382.531,A -89.96659,B 0.00000,C 180.00000} ; insert
  LIN {X 3485.893,Y 2029.899,Z -382.531,A -89.96659,B 0.00000,C 180.00000} ; release
  LIN {X 3485.893,Y 2029.899,Z -82.531,A -89.96659,B 0.00000,C 180.00000} ; retreat
  ; Step 3226, bar 1308
  LIN {X 3610.893,Y 2029.899,Z 855.478,A -89.96659,B 0.00000,C 180.00000} ; outside
  LIN {X 3610.893,Y 2029.899,Z -132.531,A -89.96659,B 0.00000,C 180.00000} ; preinsert
  LIN {X 3610.893,Y 2029.899,Z -382.531,A -89.96659,B 0.00000,C 180.00000} ; insert
  LIN {X 3610.893,Y 2029.899,Z -382.531,A -89.96659,B 0.00000,C 180.00000} ; release
  LIN {X 3610.893,Y 2029.899,Z -82.531,A -89.96659,B 0.00000,C 180.00000} ; retreat
  ; Step 3227, bar 1310
  LIN {X 3735.893,Y 2029.899,Z 855.478,A -89.96659,B 0.00000,C 180.00000} ; outside
  LIN {X 3735.893,Y 2029.899,Z -132.531,A -89.96659,B 0.00000,C 180.00000} ; preinsert
  LIN {X 3735.893,Y 2029.899,Z -382.531,A -89.96659,B 0.00000,C 180.00000} ; insert
  LIN {X 3735.893,Y 2029.899,Z -382.531,A -89.96659,B 0.00000,C 180.00000} ; release
  LIN {X 3735.893,Y 2029.899,Z -82.531,A -89.96659,B 0.00000,C 180.00000} ; retreat
  ; Step 3228, bar 1312
  LIN {X 3860.893,Y 2029.899,Z 855.478,A -89.96659,B 0.00000,C 180.00000} ; outside
  LIN {X 3860.893,Y 2029.899,Z -132.531,A -89.96659,B 0.00000,C 180.00000} ; preinsert
  LIN {X 3860.893,Y 2029.899,Z -382.531,A -89.96659,B 0.00000,C 180.00000} ; insert
  LIN {X 3860.893,Y 2029.899,Z -382.531,A -89.96659,B 0.00000,C 180.00000} ; release
  LIN {X 3860.893,Y 2029.899,Z -82.531,A -89.96659,B 0.00000,C 180.00000} ; retreat
  ; Step 3229, bar 1314
  LIN {X 3985.893,Y 2029.899,Z 855.478,A -89.96659,B 0.00000,C 180.00000} ; outside
  LIN {X 3985.893,Y 2029.899,Z -132.531,A -89.96659,B 0.00000,C 180.00000} ; preinsert
  LIN {X 3985.893,Y 2029.899,Z -382.531,A -89.96659,B 0.00000,C 180.00000} ; insert
  LIN {X 3985.893,Y 2029.899,Z -382.531,A -89.96659,B 0.00000,C 180.00000} ; release
  LIN {X 3985.893,Y 2029.899,Z -82.531,A -89.96659,B 0.00000,C 180.00000} ; retreat
  ; Step 3230, bar 1316
  LIN {X 4110.893,Y 2029.899,Z 855.478,A -89.96659,B 0.00000,C 180.00000} ; outside
  LIN {X 4110.893,Y 2029.899,Z -132.531,A -89.96659,B 0.00000,C 180.00000} ; preinsert
  LIN {X 4110.893,Y 2029.899,Z -382.531,A -89.96659,B 0.00000,C 180.00000} ; insert
  LIN {X 4110.893,Y 2029.899,Z -382.531,A -89.96659,B 0.00000,C 180.00000} ; release
  LIN {X 4110.893,Y 2029.899,Z -82.531,A -89.96659,B 0.00000,C 180.00000} ; retreat
  ; Step 3231, bar 1318
  LIN {X 4235.893,Y 2029.899,Z 855.478,A -89.96659,B 0.00000,C 180.00000} ; outside
  LIN {X 4235.893,Y 2029.899,Z -132.531,A -89.96659,B 0.00000,C 180.00000} ; preinsert
  LIN {X 4235.893,Y 2029.899,Z -382.531,A -89.96659,B 0.00000,C 180.00000} ; insert
  LIN {X 4235.893,Y 2029.899,Z -382.531,A -89.96659,B 0.00000,C 180.00000} ; release
  LIN {X 4235.893,Y 2029.899,Z -82.531,A -89.96659,B 0.00000,C 180.00000} ; retreat
  ; Step 3232, bar 1320
  LIN {X 4360.893,Y 2029.899,Z 855.478,A -89.96659,B 0.00000,C 180.00000} ; outside
  LIN {X 4360.893,Y 2029.899,Z -132.531,A -89.96659,B 0.00000,C 180.00000} ; preinsert
  LIN {X 4360.893,Y 2029.899,Z -382.531,A -89.96659,B 0.00000,C 180.00000} ; insert
  LIN {X 4360.893,Y 2029.899,Z -382.531,A -89.96659,B 0.00000,C 180.00000} ; release
  LIN {X 4360.893,Y 2029.899,Z -82.531,A -89.96659,B 0.00000,C 180.00000} ; retreat
  ; Step 3233, bar 1322
  LIN {X 4485.893,Y 2029.899,Z 855.478,A -89.96659,B 0.00000,C 180.00000} ; outside
  LIN {X 4485.893,Y 2029.899,Z -132.531,A -89.96659,B 0.00000,C 180.00000} ; preinsert
  LIN {X 4485.893,Y 2029.899,Z -382.531,A -89.96659,B 0.00000,C 180.00000} ; insert
  LIN {X 4485.893,Y 2029.899,Z -382.531,A -89.96659,B 0.00000,C 180.00000} ; release
  LIN {X 4485.893,Y 2029.899,Z -82.531,A -89.96659,B 0.00000,C 180.00000} ; retreat
  ; Step 3234, bar 1324
  LIN {X 4610.893,Y 2029.899,Z 855.478,A -89.96659,B 0.00000,C 180.00000} ; outside
  LIN {X 4610.893,Y 2029.899,Z -132.531,A -89.96659,B 0.00000,C 180.00000} ; preinsert
  LIN {X 4610.893,Y 2029.899,Z -382.531,A -89.96659,B 0.00000,C 180.00000} ; insert
  LIN {X 4610.893,Y 2029.899,Z -382.531,A -89.96659,B 0.00000,C 180.00000} ; release
  LIN {X 4610.893,Y 2029.899,Z -82.531,A -89.96659,B 0.00000,C 180.00000} ; retreat
  ; Step 3235, bar 1326
  LIN {X 4735.893,Y 2029.899,Z 855.478,A -89.96659,B 0.00000,C 180.00000} ; outside
  LIN {X 4735.893,Y 2029.899,Z -132.531,A -89.96659,B 0.00000,C 180.00000} ; preinsert
  LIN {X 4735.893,Y 2029.899,Z -382.531,A -89.96659,B 0.00000,C 180.00000} ; insert
  LIN {X 4735.893,Y 2029.899,Z -382.531,A -89.96659,B 0.00000,C 180.00000} ; release
  LIN {X 4735.893,Y 2029.899,Z -82.531,A -89.96659,B 0.00000,C 180.00000} ; retreat
  ; Step 3236, bar 1328
  LIN {X 4860.893,Y 2029.899,Z 855.478,A -89.96659,B 0.00000,C 180.00000} ; outside
  LIN {X 4860.893,Y 2029.899,Z -132.531,A -89.96659,B 0.00000,C 180.00000} ; preinsert
  LIN {X 4860.893,Y 2029.899,Z -382.531,A -89.96659,B 0.00000,C 180.00000} ; insert
  LIN {X 4860.893,Y 2029.899,Z -382.531,A -89.96659,B 0.00000,C 180.00000} ; release
  LIN {X 4860.893,Y 2029.899,Z -82.531,A -89.96659,B 0.00000,C 180.00000} ; retreat
  ; Step 3237, bar 1330
  LIN {X 4985.893,Y 2029.899,Z 855.478,A -89.96659,B 0.00000,C 180.00000} ; outside
  LIN {X 4985.893,Y 2029.899,Z -132.531,A -89.96659,B 0.00000,C 180.00000} ; preinsert
  LIN {X 4985.893,Y 2029.899,Z -382.531,A -89.96659,B 0.00000,C 180.00000} ; insert
  LIN {X 4985.893,Y 2029.899,Z -382.531,A -89.96659,B 0.00000,C 180.00000} ; release
  LIN {X 4985.893,Y 2029.899,Z -82.531,A -89.96659,B 0.00000,C 180.00000} ; retreat
  ; Step 3238, bar 1332
  LIN {X 5110.893,Y 2029.899,Z 855.478,A -89.96659,B 0.00000,C 180.00000} ; outside
  LIN {X 5110.893,Y 2029.899,Z -132.531,A -89.96659,B 0.00000,C 180.00000} ; preinsert
  LIN {X 5110.893,Y 2029.899,Z -382.531,A -89.96659,B 0.00000,C 180.00000} ; insert
  LIN {X 5110.893,Y 2029.899,Z -382.531,A -89.96659,B 0.00000,C 180.00000} ; release
  LIN {X 5110.893,Y 2029.899,Z -82.531,A -89.96659,B 0.00000,C 180.00000} ; retreat
  ; Step 3239, bar 1334
  LIN {X 5235.893,Y 2029.899,Z 855.478,A -89.96659,B 0.00000,C 180.00000} ; outside
  LIN {X 5235.893,Y 2029.899,Z -132.531,A -89.96659,B 0.00000,C 180.00000} ; preinsert
  LIN {X 5235.893,Y 2029.899,Z -382.531,A -89.96659,B 0.00000,C 180.00000} ; insert
  LIN {X 5235.893,Y 2029.899,Z -382.531,A -89.96659,B 0.00000,C 180.00000} ; release
  LIN {X 5235.893,Y 2029.899,Z -82.531,A -89.96659,B 0.00000,C 180.00000} ; retreat
  ; Step 3240, bar 1336
  LIN {X 5360.893,Y 2029.899,Z 855.478,A -89.96659,B 0.00000,C 180.00000} ; outside
  LIN {X 5360.893,Y 2029.899,Z -132.531,A -89.96659,B 0.00000,C 180.00000} ; preinsert
  LIN {X 5360.893,Y 2029.899,Z -382.531,A -89.96659,B 0.00000,C 180.00000} ; insert
  LIN {X 5360.893,Y 2029.899,Z -382.531,A -89.96659,B 0.00000,C 180.00000} ; release
  LIN {X 5360.893,Y 2029.899,Z -82.531,A -89.96659,B 0.00000,C 180.00000} ; retreat
  ; Step 3241, bar 1338
  LIN {X 5485.893,Y 2029.899,Z 855.478,A -89.96659,B 0.00000,C 180.00000} ; outside
  LIN {X 5485.893,Y 2029.899,Z -132.531,A -89.96659,B 0.00000,C 180.00000} ; preinsert
  LIN {X 5485.893,Y 2029.899,Z -382.531,A -89.96659,B 0.00000,C 180.00000} ; insert
  LIN {X 5485.893,Y 2029.899,Z -382.531,A -89.96659,B 0.00000,C 180.00000} ; release
  LIN {X 5485.893,Y 2029.899,Z -82.531,A -89.96659,B 0.00000,C 180.00000} ; retreat
  ; Step 3242, bar 1340
  LIN {X 5610.893,Y 2029.899,Z 855.478,A -89.96659,B 0.00000,C 180.00000} ; outside
  LIN {X 5610.893,Y 2029.899,Z -132.531,A -89.96659,B 0.00000,C 180.00000} ; preinsert
  LIN {X 5610.893,Y 2029.899,Z -382.531,A -89.96659,B 0.00000,C 180.00000} ; insert
  LIN {X 5610.893,Y 2029.899,Z -382.531,A -89.96659,B 0.00000,C 180.00000} ; release
  LIN {X 5610.893,Y 2029.899,Z -82.531,A -89.96659,B 0.00000,C 180.00000} ; retreat
  ; Step 3243, bar 1342
  LIN {X 5735.893,Y 2029.899,Z 855.478,A -89.96659,B 0.00000,C 180.00000} ; outside
  LIN {X 5735.893,Y 2029.899,Z -132.531,A -89.96659,B 0.00000,C 180.00000} ; preinsert
  LIN {X 5735.893,Y 2029.899,Z -382.531,A -89.96659,B 0.00000,C 180.00000} ; insert
  LIN {X 5735.893,Y 2029.899,Z -382.531,A -89.96659,B 0.00000,C 180.00000} ; release
  LIN {X 5735.893,Y 2029.899,Z -82.531,A -89.96659,B 0.00000,C 180.00000} ; retreat
  ; Step 3244, bar 1344
  LIN {X 5860.893,Y 2029.899,Z 855.478,A -89.96659,B 0.00000,C 180.00000} ; outside
  LIN {X 5860.893,Y 2029.899,Z -132.531,A -89.96659,B 0.00000,C 180.00000} ; preinsert
  LIN {X 5860.893,Y 2029.899,Z -382.531,A -89.96659,B 0.00000,C 180.00000} ; insert
  LIN {X 5860.893,Y 2029.899,Z -382.531,A -89.96659,B 0.00000,C 180.00000} ; release
  LIN {X 5860.893,Y 2029.899,Z -82.531,A -89.96659,B 0.00000,C 180.00000} ; retreat
  ; Step 3245, bar 1346
  LIN {X 6110.893,Y 2029.899,Z 855.478,A -89.96659,B 0.00000,C 180.00000} ; outside
  LIN {X 6110.893,Y 2029.899,Z -132.531,A -89.96659,B 0.00000,C 180.00000} ; preinsert
  LIN {X 6110.893,Y 2029.899,Z -382.531,A -89.96659,B 0.00000,C 180.00000} ; insert
  LIN {X 6110.893,Y 2029.899,Z -382.531,A -89.96659,B 0.00000,C 180.00000} ; release
  LIN {X 6110.893,Y 2029.899,Z -82.531,A -89.96659,B 0.00000,C 180.00000} ; retreat
  ; Step 3246, bar 1348
  LIN {X 6235.893,Y 2029.899,Z 855.478,A -89.96659,B 0.00000,C 180.00000} ; outside
  LIN {X 6235.893,Y 2029.899,Z -132.531,A -89.96659,B 0.00000,C 180.00000} ; preinsert
  LIN {X 6235.893,Y 2029.899,Z -382.531,A -89.96659,B 0.00000,C 180.00000} ; insert
  LIN {X 6235.893,Y 2029.899,Z -382.531,A -89.96659,B 0.00000,C 180.00000} ; release
  LIN {X 6235.893,Y 2029.899,Z -82.531,A -89.96659,B 0.00000,C 180.00000} ; retreat
  ; Step 3247, bar 1350
  LIN {X 6360.893,Y 2029.899,Z 855.478,A -89.96659,B 0.00000,C 180.00000} ; outside
  LIN {X 6360.893,Y 2029.899,Z -132.531,A -89.96659,B 0.00000,C 180.00000} ; preinsert
  LIN {X 6360.893,Y 2029.899,Z -382.531,A -89.96659,B 0.00000,C 180.00000} ; insert
  LIN {X 6360.893,Y 2029.899,Z -382.531,A -89.96659,B 0.00000,C 180.00000} ; release
  LIN {X 6360.893,Y 2029.899,Z -82.531,A -89.96659,B 0.00000,C 180.00000} ; retreat
  ; Step 3248, bar 1352
  LIN {X 6485.893,Y 2029.899,Z 855.478,A -89.96659,B 0.00000,C 180.00000} ; outside
  LIN {X 6485.893,Y 2029.899,Z -132.531,A -89.96659,B 0.00000,C 180.00000} ; preinsert
  LIN {X 6485.893,Y 2029.899,Z -382.531,A -89.96659,B 0.00000,C 180.00000} ; insert
  LIN {X 6485.893,Y 2029.899,Z -382.531,A -89.96659,B 0.00000,C 180.00000} ; release
  LIN {X 6485.893,Y 2029.899,Z -82.531,A -89.96659,B 0.00000,C 180.00000} ; retreat
  ; Step 3249, bar 1354
  LIN {X 6610.893,Y 2029.899,Z 855.478,A -89.96659,B 0.00000,C 180.00000} ; outside
  LIN {X 6610.893,Y 2029.899,Z -132.531,A -89.96659,B 0.00000,C 180.00000} ; preinsert
  LIN {X 6610.893,Y 2029.899,Z -382.531,A -89.96659,B 0.00000,C 180.00000} ; insert
  LIN {X 6610.893,Y 2029.899,Z -382.531,A -89.96659,B 0.00000,C 180.00000} ; release
  LIN {X 6610.893,Y 2029.899,Z -82.531,A -89.96659,B 0.00000,C 180.00000} ; retreat
  ; Step 3250, bar 1356
  LIN {X 6735.893,Y 2029.899,Z 855.478,A -89.96659,B 0.00000,C 180.00000} ; outside
  LIN {X 6735.893,Y 2029.899,Z -132.531,A -89.96659,B 0.00000,C 180.00000} ; preinsert
  LIN {X 6735.893,Y 2029.899,Z -382.531,A -89.96659,B 0.00000,C 180.00000} ; insert
  LIN {X 6735.893,Y 2029.899,Z -382.531,A -89.96659,B 0.00000,C 180.00000} ; release
  LIN {X 6735.893,Y 2029.899,Z -82.531,A -89.96659,B 0.00000,C 180.00000} ; retreat
  ; Step 3251, bar 1358
  LIN {X 6860.893,Y 2029.899,Z 855.478,A -89.96659,B 0.00000,C 180.00000} ; outside
  LIN {X 6860.893,Y 2029.899,Z -132.531,A -89.96659,B 0.00000,C 180.00000} ; preinsert
  LIN {X 6860.893,Y 2029.899,Z -382.531,A -89.96659,B 0.00000,C 180.00000} ; insert
  LIN {X 6860.893,Y 2029.899,Z -382.531,A -89.96659,B 0.00000,C 180.00000} ; release
  LIN {X 6860.893,Y 2029.899,Z -82.531,A -89.96659,B 0.00000,C 180.00000} ; retreat
  ; Step 3252, bar 1360
  LIN {X 6985.893,Y 2029.899,Z 855.478,A -89.96659,B 0.00000,C 180.00000} ; outside
  LIN {X 6985.893,Y 2029.899,Z -132.531,A -89.96659,B 0.00000,C 180.00000} ; preinsert
  LIN {X 6985.893,Y 2029.899,Z -382.531,A -89.96659,B 0.00000,C 180.00000} ; insert
  LIN {X 6985.893,Y 2029.899,Z -382.531,A -89.96659,B 0.00000,C 180.00000} ; release
  LIN {X 6985.893,Y 2029.899,Z -82.531,A -89.96659,B 0.00000,C 180.00000} ; retreat
  ; Step 3253, bar 1362
  LIN {X 7110.893,Y 2029.899,Z 855.478,A -89.96659,B 0.00000,C 180.00000} ; outside
  LIN {X 7110.893,Y 2029.899,Z -132.531,A -89.96659,B 0.00000,C 180.00000} ; preinsert
  LIN {X 7110.893,Y 2029.899,Z -382.531,A -89.96659,B 0.00000,C 180.00000} ; insert
  LIN {X 7110.893,Y 2029.899,Z -382.531,A -89.96659,B 0.00000,C 180.00000} ; release
  LIN {X 7110.893,Y 2029.899,Z -82.531,A -89.96659,B 0.00000,C 180.00000} ; retreat
  ; Step 3254, bar 1364
  LIN {X 7235.893,Y 2029.899,Z 855.478,A -89.96659,B 0.00000,C 180.00000} ; outside
  LIN {X 7235.893,Y 2029.899,Z -132.531,A -89.96659,B 0.00000,C 180.00000} ; preinsert
  LIN {X 7235.893,Y 2029.899,Z -382.531,A -89.96659,B 0.00000,C 180.00000} ; insert
  LIN {X 7235.893,Y 2029.899,Z -382.531,A -89.96659,B 0.00000,C 180.00000} ; release
  LIN {X 7235.893,Y 2029.899,Z -82.531,A -89.96659,B 0.00000,C 180.00000} ; retreat
  ; Step 3255, bar 1366
  LIN {X 7360.893,Y 2029.899,Z 855.478,A -89.96659,B 0.00000,C 180.00000} ; outside
  LIN {X 7360.893,Y 2029.899,Z -132.531,A -89.96659,B 0.00000,C 180.00000} ; preinsert
  LIN {X 7360.893,Y 2029.899,Z -382.531,A -89.96659,B 0.00000,C 180.00000} ; insert
  LIN {X 7360.893,Y 2029.899,Z -382.531,A -89.96659,B 0.00000,C 180.00000} ; release
  LIN {X 7360.893,Y 2029.899,Z -82.531,A -89.96659,B 0.00000,C 180.00000} ; retreat
  ; Step 3256, bar 1368
  LIN {X 7485.893,Y 2029.899,Z 855.478,A -89.96659,B 0.00000,C 180.00000} ; outside
  LIN {X 7485.893,Y 2029.899,Z -132.531,A -89.96659,B 0.00000,C 180.00000} ; preinsert
  LIN {X 7485.893,Y 2029.899,Z -382.531,A -89.96659,B 0.00000,C 180.00000} ; insert
  LIN {X 7485.893,Y 2029.899,Z -382.531,A -89.96659,B 0.00000,C 180.00000} ; release
  LIN {X 7485.893,Y 2029.899,Z -82.531,A -89.96659,B 0.00000,C 180.00000} ; retreat
  ; Step 3257, bar 1370
  LIN {X 7610.893,Y 2029.899,Z 855.478,A -89.96659,B 0.00000,C 180.00000} ; outside
  LIN {X 7610.893,Y 2029.899,Z -132.531,A -89.96659,B 0.00000,C 180.00000} ; preinsert
  LIN {X 7610.893,Y 2029.899,Z -382.531,A -89.96659,B 0.00000,C 180.00000} ; insert
  LIN {X 7610.893,Y 2029.899,Z -382.531,A -89.96659,B 0.00000,C 180.00000} ; release
  LIN {X 7610.893,Y 2029.899,Z -82.531,A -89.96659,B 0.00000,C 180.00000} ; retreat
  ; Step 3258, bar 1372
  LIN {X 7735.893,Y 2029.899,Z 855.478,A -89.96659,B 0.00000,C 180.00000} ; outside
  LIN {X 7735.893,Y 2029.899,Z -132.531,A -89.96659,B 0.00000,C 180.00000} ; preinsert
  LIN {X 7735.893,Y 2029.899,Z -382.531,A -89.96659,B 0.00000,C 180.00000} ; insert
  LIN {X 7735.893,Y 2029.899,Z -382.531,A -89.96659,B 0.00000,C 180.00000} ; release
  LIN {X 7735.893,Y 2029.899,Z -82.531,A -89.96659,B 0.00000,C 180.00000} ; retreat
  ; Step 3259, bar 1374
  LIN {X 7860.893,Y 2029.899,Z 855.478,A -89.96659,B 0.00000,C 180.00000} ; outside
  LIN {X 7860.893,Y 2029.899,Z -132.531,A -89.96659,B 0.00000,C 180.00000} ; preinsert
  LIN {X 7860.893,Y 2029.899,Z -382.531,A -89.96659,B 0.00000,C 180.00000} ; insert
  LIN {X 7860.893,Y 2029.899,Z -382.531,A -89.96659,B 0.00000,C 180.00000} ; release
  LIN {X 7860.893,Y 2029.899,Z -82.531,A -89.96659,B 0.00000,C 180.00000} ; retreat
  ; Step 3260, bar 1376
  LIN {X 7985.893,Y 2029.899,Z 855.478,A -89.96659,B 0.00000,C 180.00000} ; outside
  LIN {X 7985.893,Y 2029.899,Z -132.531,A -89.96659,B 0.00000,C 180.00000} ; preinsert
  LIN {X 7985.893,Y 2029.899,Z -382.531,A -89.96659,B 0.00000,C 180.00000} ; insert
  LIN {X 7985.893,Y 2029.899,Z -382.531,A -89.96659,B 0.00000,C 180.00000} ; release
  LIN {X 7985.893,Y 2029.899,Z -82.531,A -89.96659,B 0.00000,C 180.00000} ; retreat
  ; Step 3261, bar 1378
  LIN {X 8110.893,Y 2029.899,Z 855.478,A -89.96659,B 0.00000,C 180.00000} ; outside
  LIN {X 8110.893,Y 2029.899,Z -132.531,A -89.96659,B 0.00000,C 180.00000} ; preinsert
  LIN {X 8110.893,Y 2029.899,Z -382.531,A -89.96659,B 0.00000,C 180.00000} ; insert
  LIN {X 8110.893,Y 2029.899,Z -382.531,A -89.96659,B 0.00000,C 180.00000} ; release
  LIN {X 8110.893,Y 2029.899,Z -82.531,A -89.96659,B 0.00000,C 180.00000} ; retreat
  ; Step 3262, bar 1380
  LIN {X 8235.893,Y 2029.899,Z 855.478,A -89.96659,B 0.00000,C -180.00000} ; outside
  LIN {X 8235.893,Y 2029.899,Z -132.531,A -89.96659,B 0.00000,C -180.00000} ; preinsert
  LIN {X 8235.893,Y 2029.899,Z -382.531,A -89.96659,B 0.00000,C -180.00000} ; insert
  LIN {X 8235.893,Y 2029.899,Z -382.531,A -89.96659,B 0.00000,C -180.00000} ; release
  LIN {X 8235.893,Y 2029.899,Z -82.531,A -89.96659,B 0.00000,C -180.00000} ; retreat
  ; Step 3263, bar 1382
  LIN {X 8360.893,Y 2029.899,Z 855.478,A -89.96659,B 0.00000,C -180.00000} ; outside
  LIN {X 8360.893,Y 2029.899,Z -132.531,A -89.96659,B 0.00000,C -180.00000} ; preinsert
  LIN {X 8360.893,Y 2029.899,Z -382.531,A -89.96659,B 0.00000,C -180.00000} ; insert
  LIN {X 8360.893,Y 2029.899,Z -382.531,A -89.96659,B 0.00000,C -180.00000} ; release
  LIN {X 8360.893,Y 2029.899,Z -82.531,A -89.96659,B 0.00000,C -180.00000} ; retreat
  ; Step 3264, bar 1384
  LIN {X 8485.893,Y 2029.899,Z 855.478,A -89.96659,B 0.00000,C -180.00000} ; outside
  LIN {X 8485.893,Y 2029.899,Z -132.531,A -89.96659,B 0.00000,C -180.00000} ; preinsert
  LIN {X 8485.893,Y 2029.899,Z -382.531,A -89.96659,B 0.00000,C -180.00000} ; insert
  LIN {X 8485.893,Y 2029.899,Z -382.531,A -89.96659,B 0.00000,C -180.00000} ; release
  LIN {X 8485.893,Y 2029.899,Z -82.531,A -89.96659,B 0.00000,C -180.00000} ; retreat
  ; Step 3265, bar 1386
  LIN {X 8610.893,Y 2029.899,Z 855.478,A -89.96659,B 0.00000,C -180.00000} ; outside
  LIN {X 8610.893,Y 2029.899,Z -132.531,A -89.96659,B 0.00000,C -180.00000} ; preinsert
  LIN {X 8610.893,Y 2029.899,Z -382.531,A -89.96659,B 0.00000,C -180.00000} ; insert
  LIN {X 8610.893,Y 2029.899,Z -382.531,A -89.96659,B 0.00000,C -180.00000} ; release
  LIN {X 8610.893,Y 2029.899,Z -82.531,A -89.96659,B 0.00000,C -180.00000} ; retreat
  ; Step 3266, bar 1388
  LIN {X 8735.893,Y 2029.899,Z 855.478,A -89.96659,B 0.00000,C -180.00000} ; outside
  LIN {X 8735.893,Y 2029.899,Z -132.531,A -89.96659,B 0.00000,C -180.00000} ; preinsert
  LIN {X 8735.893,Y 2029.899,Z -382.531,A -89.96659,B 0.00000,C -180.00000} ; insert
  LIN {X 8735.893,Y 2029.899,Z -382.531,A -89.96659,B 0.00000,C -180.00000} ; release
  LIN {X 8735.893,Y 2029.899,Z -82.531,A -89.96659,B 0.00000,C -180.00000} ; retreat
  ; Step 3267, bar 1390
  LIN {X 8860.893,Y 2029.899,Z 855.478,A -89.96659,B 0.00000,C -180.00000} ; outside
  LIN {X 8860.893,Y 2029.899,Z -132.531,A -89.96659,B 0.00000,C -180.00000} ; preinsert
  LIN {X 8860.893,Y 2029.899,Z -382.531,A -89.96659,B 0.00000,C -180.00000} ; insert
  LIN {X 8860.893,Y 2029.899,Z -382.531,A -89.96659,B 0.00000,C -180.00000} ; release
  LIN {X 8860.893,Y 2029.899,Z -82.531,A -89.96659,B 0.00000,C -180.00000} ; retreat
  ; Step 3268, bar 1392
  LIN {X 8985.893,Y 2029.899,Z 855.478,A -89.96659,B 0.00000,C -180.00000} ; outside
  LIN {X 8985.893,Y 2029.899,Z -132.531,A -89.96659,B 0.00000,C -180.00000} ; preinsert
  LIN {X 8985.893,Y 2029.899,Z -382.531,A -89.96659,B 0.00000,C -180.00000} ; insert
  LIN {X 8985.893,Y 2029.899,Z -382.531,A -89.96659,B 0.00000,C -180.00000} ; release
  LIN {X 8985.893,Y 2029.899,Z -82.531,A -89.96659,B 0.00000,C -180.00000} ; retreat
  ; Step 3269, bar 1394
  LIN {X 9110.893,Y 2029.899,Z 855.478,A -89.96659,B 0.00000,C -180.00000} ; outside
  LIN {X 9110.893,Y 2029.899,Z -132.531,A -89.96659,B 0.00000,C -180.00000} ; preinsert
  LIN {X 9110.893,Y 2029.899,Z -382.531,A -89.96659,B 0.00000,C -180.00000} ; insert
  LIN {X 9110.893,Y 2029.899,Z -382.531,A -89.96659,B 0.00000,C -180.00000} ; release
  LIN {X 9110.893,Y 2029.899,Z -82.531,A -89.96659,B 0.00000,C -180.00000} ; retreat
  ; Step 3270, bar 1396
  LIN {X 9235.893,Y 2029.899,Z 855.478,A -89.96659,B 0.00000,C -180.00000} ; outside
  LIN {X 9235.893,Y 2029.899,Z -132.531,A -89.96659,B 0.00000,C -180.00000} ; preinsert
  LIN {X 9235.893,Y 2029.899,Z -382.531,A -89.96659,B 0.00000,C -180.00000} ; insert
  LIN {X 9235.893,Y 2029.899,Z -382.531,A -89.96659,B 0.00000,C -180.00000} ; release
  LIN {X 9235.893,Y 2029.899,Z -82.531,A -89.96659,B 0.00000,C -180.00000} ; retreat
  ; Step 3271, bar 1398
  LIN {X 9360.893,Y 2029.899,Z 855.478,A -89.96659,B 0.00000,C -180.00000} ; outside
  LIN {X 9360.893,Y 2029.899,Z -132.531,A -89.96659,B 0.00000,C -180.00000} ; preinsert
  LIN {X 9360.893,Y 2029.899,Z -382.531,A -89.96659,B 0.00000,C -180.00000} ; insert
  LIN {X 9360.893,Y 2029.899,Z -382.531,A -89.96659,B 0.00000,C -180.00000} ; release
  LIN {X 9360.893,Y 2029.899,Z -82.531,A -89.96659,B 0.00000,C -180.00000} ; retreat
  ; Step 3272, bar 1400
  LIN {X 9485.893,Y 2029.899,Z 855.478,A -89.96659,B 0.00000,C -180.00000} ; outside
  LIN {X 9485.893,Y 2029.899,Z -132.531,A -89.96659,B 0.00000,C -180.00000} ; preinsert
  LIN {X 9485.893,Y 2029.899,Z -382.531,A -89.96659,B 0.00000,C -180.00000} ; insert
  LIN {X 9485.893,Y 2029.899,Z -382.531,A -89.96659,B 0.00000,C -180.00000} ; release
  LIN {X 9485.893,Y 2029.899,Z -82.531,A -89.96659,B 0.00000,C -180.00000} ; retreat
  ; Step 3273, bar 1402
  LIN {X 9610.893,Y 2029.899,Z 855.478,A -89.96659,B 0.00000,C -180.00000} ; outside
  LIN {X 9610.893,Y 2029.899,Z -132.531,A -89.96659,B 0.00000,C -180.00000} ; preinsert
  LIN {X 9610.893,Y 2029.899,Z -382.531,A -89.96659,B 0.00000,C -180.00000} ; insert
  LIN {X 9610.893,Y 2029.899,Z -382.531,A -89.96659,B 0.00000,C -180.00000} ; release
  LIN {X 9610.893,Y 2029.899,Z -82.531,A -89.96659,B 0.00000,C -180.00000} ; retreat
  ; Step 3274, bar 1404
  LIN {X 9735.893,Y 2029.899,Z 855.478,A -89.96659,B 0.00000,C -180.00000} ; outside
  LIN {X 9735.893,Y 2029.899,Z -132.531,A -89.96659,B 0.00000,C -180.00000} ; preinsert
  LIN {X 9735.893,Y 2029.899,Z -382.531,A -89.96659,B 0.00000,C -180.00000} ; insert
  LIN {X 9735.893,Y 2029.899,Z -382.531,A -89.96659,B 0.00000,C -180.00000} ; release
  LIN {X 9735.893,Y 2029.899,Z -82.531,A -89.96659,B 0.00000,C -180.00000} ; retreat
  ; Step 3275, bar 1406
  LIN {X 9860.893,Y 2029.899,Z 855.478,A -89.96659,B 0.00000,C -180.00000} ; outside
  LIN {X 9860.893,Y 2029.899,Z -132.531,A -89.96659,B 0.00000,C -180.00000} ; preinsert
  LIN {X 9860.893,Y 2029.899,Z -382.531,A -89.96659,B 0.00000,C -180.00000} ; insert
  LIN {X 9860.893,Y 2029.899,Z -382.531,A -89.96659,B 0.00000,C -180.00000} ; release
  LIN {X 9860.893,Y 2029.899,Z -82.531,A -89.96659,B 0.00000,C -180.00000} ; retreat
  ; Step 3276, bar 1408
  LIN {X 10110.893,Y 2029.899,Z 855.478,A -89.96659,B 0.00000,C -180.00000} ; outside
  LIN {X 10110.893,Y 2029.899,Z -132.531,A -89.96659,B 0.00000,C -180.00000} ; preinsert
  LIN {X 10110.893,Y 2029.899,Z -382.531,A -89.96659,B 0.00000,C -180.00000} ; insert
  LIN {X 10110.893,Y 2029.899,Z -382.531,A -89.96659,B 0.00000,C -180.00000} ; release
  LIN {X 10110.893,Y 2029.899,Z -82.531,A -89.96659,B 0.00000,C -180.00000} ; retreat
  ; Step 3277, bar 1410
  LIN {X 10235.893,Y 2029.899,Z 855.478,A -89.96659,B 0.00000,C -180.00000} ; outside
  LIN {X 10235.893,Y 2029.899,Z -132.531,A -89.96659,B 0.00000,C -180.00000} ; preinsert
  LIN {X 10235.893,Y 2029.899,Z -382.531,A -89.96659,B 0.00000,C -180.00000} ; insert
  LIN {X 10235.893,Y 2029.899,Z -382.531,A -89.96659,B 0.00000,C -180.00000} ; release
  LIN {X 10235.893,Y 2029.899,Z -82.531,A -89.96659,B 0.00000,C -180.00000} ; retreat
  ; Step 3278, bar 1412
  LIN {X 10360.893,Y 2029.899,Z 855.478,A -89.96659,B 0.00000,C -180.00000} ; outside
  LIN {X 10360.893,Y 2029.899,Z -132.531,A -89.96659,B 0.00000,C -180.00000} ; preinsert
  LIN {X 10360.893,Y 2029.899,Z -382.531,A -89.96659,B 0.00000,C -180.00000} ; insert
  LIN {X 10360.893,Y 2029.899,Z -382.531,A -89.96659,B 0.00000,C -180.00000} ; release
  LIN {X 10360.893,Y 2029.899,Z -82.531,A -89.96659,B 0.00000,C -180.00000} ; retreat
  ; Step 3279, bar 1414
  LIN {X 10485.893,Y 2029.899,Z 855.478,A -89.96659,B 0.00000,C -180.00000} ; outside
  LIN {X 10485.893,Y 2029.899,Z -132.531,A -89.96659,B 0.00000,C -180.00000} ; preinsert
  LIN {X 10485.893,Y 2029.899,Z -382.531,A -89.96659,B 0.00000,C -180.00000} ; insert
  LIN {X 10485.893,Y 2029.899,Z -382.531,A -89.96659,B 0.00000,C -180.00000} ; release
  LIN {X 10485.893,Y 2029.899,Z -82.531,A -89.96659,B 0.00000,C -180.00000} ; retreat
  ; Step 3280, bar 1416
  LIN {X 10610.893,Y 2029.899,Z 855.478,A -89.96659,B 0.00000,C -180.00000} ; outside
  LIN {X 10610.893,Y 2029.899,Z -132.531,A -89.96659,B 0.00000,C -180.00000} ; preinsert
  LIN {X 10610.893,Y 2029.899,Z -382.531,A -89.96659,B 0.00000,C -180.00000} ; insert
  LIN {X 10610.893,Y 2029.899,Z -382.531,A -89.96659,B 0.00000,C -180.00000} ; release
  LIN {X 10610.893,Y 2029.899,Z -82.531,A -89.96659,B 0.00000,C -180.00000} ; retreat
  ; Step 3281, bar 1418
  LIN {X 10735.893,Y 2029.899,Z 855.478,A -89.96659,B 0.00000,C -180.00000} ; outside
  LIN {X 10735.893,Y 2029.899,Z -132.531,A -89.96659,B 0.00000,C -180.00000} ; preinsert
  LIN {X 10735.893,Y 2029.899,Z -382.531,A -89.96659,B 0.00000,C -180.00000} ; insert
  LIN {X 10735.893,Y 2029.899,Z -382.531,A -89.96659,B 0.00000,C -180.00000} ; release
  LIN {X 10735.893,Y 2029.899,Z -82.531,A -89.96659,B 0.00000,C -180.00000} ; retreat
  ; Step 3282, bar 1420
  LIN {X 10860.893,Y 2029.899,Z 855.478,A -89.96659,B 0.00000,C -180.00000} ; outside
  LIN {X 10860.893,Y 2029.899,Z -132.531,A -89.96659,B 0.00000,C -180.00000} ; preinsert
  LIN {X 10860.893,Y 2029.899,Z -382.531,A -89.96659,B 0.00000,C -180.00000} ; insert
  LIN {X 10860.893,Y 2029.899,Z -382.531,A -89.96659,B 0.00000,C -180.00000} ; release
  LIN {X 10860.893,Y 2029.899,Z -82.531,A -89.96659,B 0.00000,C -180.00000} ; retreat
  ; Step 3283, bar 1422
  LIN {X 10985.893,Y 2029.899,Z 855.478,A -89.96659,B 0.00000,C -180.00000} ; outside
  LIN {X 10985.893,Y 2029.899,Z -132.531,A -89.96659,B 0.00000,C -180.00000} ; preinsert
  LIN {X 10985.893,Y 2029.899,Z -382.531,A -89.96659,B 0.00000,C -180.00000} ; insert
  LIN {X 10985.893,Y 2029.899,Z -382.531,A -89.96659,B 0.00000,C -180.00000} ; release
  LIN {X 10985.893,Y 2029.899,Z -82.531,A -89.96659,B 0.00000,C -180.00000} ; retreat
  ; Step 3284, bar 1424
  LIN {X 11110.893,Y 2029.899,Z 855.478,A -89.96659,B 0.00000,C -180.00000} ; outside
  LIN {X 11110.893,Y 2029.899,Z -132.531,A -89.96659,B 0.00000,C -180.00000} ; preinsert
  LIN {X 11110.893,Y 2029.899,Z -382.531,A -89.96659,B 0.00000,C -180.00000} ; insert
  LIN {X 11110.893,Y 2029.899,Z -382.531,A -89.96659,B 0.00000,C -180.00000} ; release
  LIN {X 11110.893,Y 2029.899,Z -82.531,A -89.96659,B 0.00000,C -180.00000} ; retreat
  ; Step 3285, bar 1426
  LIN {X 11235.893,Y 2029.899,Z 855.478,A -89.96659,B 0.00000,C -180.00000} ; outside
  LIN {X 11235.893,Y 2029.899,Z -132.531,A -89.96659,B 0.00000,C -180.00000} ; preinsert
  LIN {X 11235.893,Y 2029.899,Z -382.531,A -89.96659,B 0.00000,C -180.00000} ; insert
  LIN {X 11235.893,Y 2029.899,Z -382.531,A -89.96659,B 0.00000,C -180.00000} ; release
  LIN {X 11235.893,Y 2029.899,Z -82.531,A -89.96659,B 0.00000,C -180.00000} ; retreat
  ; Step 3286, bar 1428
  LIN {X 11360.893,Y 2029.899,Z 855.478,A -89.96659,B 0.00000,C -180.00000} ; outside
  LIN {X 11360.893,Y 2029.899,Z -132.531,A -89.96659,B 0.00000,C -180.00000} ; preinsert
  LIN {X 11360.893,Y 2029.899,Z -382.531,A -89.96659,B 0.00000,C -180.00000} ; insert
  LIN {X 11360.893,Y 2029.899,Z -382.531,A -89.96659,B 0.00000,C -180.00000} ; release
  LIN {X 11360.893,Y 2029.899,Z -82.531,A -89.96659,B 0.00000,C -180.00000} ; retreat
  ; Step 3287, bar 1430
  LIN {X 11485.893,Y 2029.899,Z 855.478,A -89.96659,B 0.00000,C -180.00000} ; outside
  LIN {X 11485.893,Y 2029.899,Z -132.531,A -89.96659,B 0.00000,C -180.00000} ; preinsert
  LIN {X 11485.893,Y 2029.899,Z -382.531,A -89.96659,B 0.00000,C -180.00000} ; insert
  LIN {X 11485.893,Y 2029.899,Z -382.531,A -89.96659,B 0.00000,C -180.00000} ; release
  LIN {X 11485.893,Y 2029.899,Z -82.531,A -89.96659,B 0.00000,C -180.00000} ; retreat
  ; Step 3288, bar 1432
  LIN {X 11610.893,Y 2029.899,Z 855.478,A -89.96659,B 0.00000,C -180.00000} ; outside
  LIN {X 11610.893,Y 2029.899,Z -132.531,A -89.96659,B 0.00000,C -180.00000} ; preinsert
  LIN {X 11610.893,Y 2029.899,Z -382.531,A -89.96659,B 0.00000,C -180.00000} ; insert
  LIN {X 11610.893,Y 2029.899,Z -382.531,A -89.96659,B 0.00000,C -180.00000} ; release
  LIN {X 11610.893,Y 2029.899,Z -82.531,A -89.96659,B 0.00000,C -180.00000} ; retreat
  ; Step 3289, bar 1434
  LIN {X 11735.893,Y 2029.899,Z 855.478,A -89.96659,B 0.00000,C -180.00000} ; outside
  LIN {X 11735.893,Y 2029.899,Z -132.531,A -89.96659,B 0.00000,C -180.00000} ; preinsert
  LIN {X 11735.893,Y 2029.899,Z -382.531,A -89.96659,B 0.00000,C -180.00000} ; insert
  LIN {X 11735.893,Y 2029.899,Z -382.531,A -89.96659,B 0.00000,C -180.00000} ; release
  LIN {X 11735.893,Y 2029.899,Z -82.531,A -89.96659,B 0.00000,C -180.00000} ; retreat
  ; Step 3290, bar 1436
  LIN {X 11860.893,Y 2029.899,Z 855.478,A -89.96659,B 0.00000,C -180.00000} ; outside
  LIN {X 11860.893,Y 2029.899,Z -132.531,A -89.96659,B 0.00000,C -180.00000} ; preinsert
  LIN {X 11860.893,Y 2029.899,Z -382.531,A -89.96659,B 0.00000,C -180.00000} ; insert
  LIN {X 11860.893,Y 2029.899,Z -382.531,A -89.96659,B 0.00000,C -180.00000} ; release
  LIN {X 11860.893,Y 2029.899,Z -82.531,A -89.96659,B 0.00000,C -180.00000} ; retreat
  ; Step 3291, bar 1438
  LIN {X 11985.893,Y 2029.899,Z 855.478,A -89.96659,B 0.00000,C -180.00000} ; outside
  LIN {X 11985.893,Y 2029.899,Z -132.531,A -89.96659,B 0.00000,C -180.00000} ; preinsert
  LIN {X 11985.893,Y 2029.899,Z -382.531,A -89.96659,B 0.00000,C -180.00000} ; insert
  LIN {X 11985.893,Y 2029.899,Z -382.531,A -89.96659,B 0.00000,C -180.00000} ; release
  LIN {X 11985.893,Y 2029.899,Z -82.531,A -89.96659,B 0.00000,C -180.00000} ; retreat
  ; Step 3292, bar 1440
  LIN {X 12110.893,Y 2029.899,Z 855.478,A -89.96659,B 0.00000,C -180.00000} ; outside
  LIN {X 12110.893,Y 2029.899,Z -132.531,A -89.96659,B 0.00000,C -180.00000} ; preinsert
  LIN {X 12110.893,Y 2029.899,Z -382.531,A -89.96659,B 0.00000,C -180.00000} ; insert
  LIN {X 12110.893,Y 2029.899,Z -382.531,A -89.96659,B 0.00000,C -180.00000} ; release
  LIN {X 12110.893,Y 2029.899,Z -82.531,A -89.96659,B 0.00000,C -180.00000} ; retreat
  ; Step 3293, bar 1442
  LIN {X 12235.893,Y 2029.899,Z 855.478,A -89.96659,B 0.00000,C -180.00000} ; outside
  LIN {X 12235.893,Y 2029.899,Z -132.531,A -89.96659,B 0.00000,C -180.00000} ; preinsert
  LIN {X 12235.893,Y 2029.899,Z -382.531,A -89.96659,B 0.00000,C -180.00000} ; insert
  LIN {X 12235.893,Y 2029.899,Z -382.531,A -89.96659,B 0.00000,C -180.00000} ; release
  LIN {X 12235.893,Y 2029.899,Z -82.531,A -89.96659,B 0.00000,C -180.00000} ; retreat
  ; Step 3294, bar 1444
  LIN {X 12335.893,Y 2029.899,Z 855.478,A -89.96659,B 0.00000,C -180.00000} ; outside
  LIN {X 12335.893,Y 2029.899,Z -132.531,A -89.96659,B 0.00000,C -180.00000} ; preinsert
  LIN {X 12335.893,Y 2029.899,Z -382.531,A -89.96659,B 0.00000,C -180.00000} ; insert
  LIN {X 12335.893,Y 2029.899,Z -382.531,A -89.96659,B 0.00000,C -180.00000} ; release
  LIN {X 12335.893,Y 2029.899,Z -82.531,A -89.96659,B 0.00000,C -180.00000} ; retreat
  ; Step 3295, bar 1446
  LIN {X 12435.893,Y 2029.899,Z 855.478,A -89.96659,B 0.00000,C -180.00000} ; outside
  LIN {X 12435.893,Y 2029.899,Z -132.531,A -89.96659,B 0.00000,C -180.00000} ; preinsert
  LIN {X 12435.893,Y 2029.899,Z -382.531,A -89.96659,B 0.00000,C -180.00000} ; insert
  LIN {X 12435.893,Y 2029.899,Z -382.531,A -89.96659,B 0.00000,C -180.00000} ; release
  LIN {X 12435.893,Y 2029.899,Z -82.531,A -89.96659,B 0.00000,C -180.00000} ; retreat
  ; Step 3296, bar 1448
  LIN {X 12535.893,Y 2029.899,Z 855.478,A -89.96659,B 0.00000,C -180.00000} ; outside
  LIN {X 12535.893,Y 2029.899,Z -132.531,A -89.96659,B 0.00000,C -180.00000} ; preinsert
  LIN {X 12535.893,Y 2029.899,Z -382.531,A -89.96659,B 0.00000,C -180.00000} ; insert
  LIN {X 12535.893,Y 2029.899,Z -382.531,A -89.96659,B 0.00000,C -180.00000} ; release
  LIN {X 12535.893,Y 2029.899,Z -82.531,A -89.96659,B 0.00000,C -180.00000} ; retreat
  ; Step 3297, bar 1450
  LIN {X 12635.893,Y 2029.899,Z 855.478,A -89.96659,B 0.00000,C -180.00000} ; outside
  LIN {X 12635.893,Y 2029.899,Z -132.531,A -89.96659,B 0.00000,C -180.00000} ; preinsert
  LIN {X 12635.893,Y 2029.899,Z -382.531,A -89.96659,B 0.00000,C -180.00000} ; insert
  LIN {X 12635.893,Y 2029.899,Z -382.531,A -89.96659,B 0.00000,C -180.00000} ; release
  LIN {X 12635.893,Y 2029.899,Z -82.531,A -89.96659,B 0.00000,C -180.00000} ; retreat
  ; Step 3298, bar 1452
  LIN {X 12735.893,Y 2029.899,Z 855.478,A -89.96659,B 0.00000,C -180.00000} ; outside
  LIN {X 12735.893,Y 2029.899,Z -132.531,A -89.96659,B 0.00000,C -180.00000} ; preinsert
  LIN {X 12735.893,Y 2029.899,Z -382.531,A -89.96659,B 0.00000,C -180.00000} ; insert
  LIN {X 12735.893,Y 2029.899,Z -382.531,A -89.96659,B 0.00000,C -180.00000} ; release
  LIN {X 12735.893,Y 2029.899,Z -82.531,A -89.96659,B 0.00000,C -180.00000} ; retreat
  ; Step 3299, bar 1454
  LIN {X 12835.893,Y 2029.899,Z 855.478,A -89.96659,B 0.00000,C -180.00000} ; outside
  LIN {X 12835.893,Y 2029.899,Z -132.531,A -89.96659,B 0.00000,C -180.00000} ; preinsert
  LIN {X 12835.893,Y 2029.899,Z -382.531,A -89.96659,B 0.00000,C -180.00000} ; insert
  LIN {X 12835.893,Y 2029.899,Z -382.531,A -89.96659,B 0.00000,C -180.00000} ; release
  LIN {X 12835.893,Y 2029.899,Z -82.531,A -89.96659,B 0.00000,C -180.00000} ; retreat
  ; Step 3300, bar 1456
  LIN {X 12935.893,Y 2029.899,Z 855.478,A -89.96659,B 0.00000,C -180.00000} ; outside
  LIN {X 12935.893,Y 2029.899,Z -132.531,A -89.96659,B 0.00000,C -180.00000} ; preinsert
  LIN {X 12935.893,Y 2029.899,Z -382.531,A -89.96659,B 0.00000,C -180.00000} ; insert
  LIN {X 12935.893,Y 2029.899,Z -382.531,A -89.96659,B 0.00000,C -180.00000} ; release
  LIN {X 12935.893,Y 2029.899,Z -82.531,A -89.96659,B 0.00000,C -180.00000} ; retreat
  ; Step 3301, bar 1458
  LIN {X 13035.893,Y 2029.899,Z 855.478,A -89.96659,B 0.00000,C -180.00000} ; outside
  LIN {X 13035.893,Y 2029.899,Z -132.531,A -89.96659,B 0.00000,C -180.00000} ; preinsert
  LIN {X 13035.893,Y 2029.899,Z -382.531,A -89.96659,B 0.00000,C -180.00000} ; insert
  LIN {X 13035.893,Y 2029.899,Z -382.531,A -89.96659,B 0.00000,C -180.00000} ; release
  LIN {X 13035.893,Y 2029.899,Z -82.531,A -89.96659,B 0.00000,C -180.00000} ; retreat
  ; Step 3302, bar 1460
  LIN {X 13135.893,Y 2029.899,Z 855.478,A -89.96659,B 0.00000,C -180.00000} ; outside
  LIN {X 13135.893,Y 2029.899,Z -132.531,A -89.96659,B 0.00000,C -180.00000} ; preinsert
  LIN {X 13135.893,Y 2029.899,Z -382.531,A -89.96659,B 0.00000,C -180.00000} ; insert
  LIN {X 13135.893,Y 2029.899,Z -382.531,A -89.96659,B 0.00000,C -180.00000} ; release
  LIN {X 13135.893,Y 2029.899,Z -82.531,A -89.96659,B 0.00000,C -180.00000} ; retreat
  ; Step 3303, bar 1462
  LIN {X 13235.893,Y 2029.899,Z 855.478,A -89.96659,B 0.00000,C -180.00000} ; outside
  LIN {X 13235.893,Y 2029.899,Z -132.531,A -89.96659,B 0.00000,C -180.00000} ; preinsert
  LIN {X 13235.893,Y 2029.899,Z -382.531,A -89.96659,B 0.00000,C -180.00000} ; insert
  LIN {X 13235.893,Y 2029.899,Z -382.531,A -89.96659,B 0.00000,C -180.00000} ; release
  LIN {X 13235.893,Y 2029.899,Z -82.531,A -89.96659,B 0.00000,C -180.00000} ; retreat
  ; Step 3304, bar 1464
  LIN {X 13335.893,Y 2029.899,Z 855.478,A -89.96659,B 0.00000,C -180.00000} ; outside
  LIN {X 13335.893,Y 2029.899,Z -132.531,A -89.96659,B 0.00000,C -180.00000} ; preinsert
  LIN {X 13335.893,Y 2029.899,Z -382.531,A -89.96659,B 0.00000,C -180.00000} ; insert
  LIN {X 13335.893,Y 2029.899,Z -382.531,A -89.96659,B 0.00000,C -180.00000} ; release
  LIN {X 13335.893,Y 2029.899,Z -82.531,A -89.96659,B 0.00000,C -180.00000} ; retreat
  ; Step 3305, bar 1466
  LIN {X 13435.893,Y 2029.899,Z 855.478,A -89.96659,B 0.00000,C -180.00000} ; outside
  LIN {X 13435.893,Y 2029.899,Z -132.531,A -89.96659,B 0.00000,C -180.00000} ; preinsert
  LIN {X 13435.893,Y 2029.899,Z -382.531,A -89.96659,B 0.00000,C -180.00000} ; insert
  LIN {X 13435.893,Y 2029.899,Z -382.531,A -89.96659,B 0.00000,C -180.00000} ; release
  LIN {X 13435.893,Y 2029.899,Z -82.531,A -89.96659,B 0.00000,C -180.00000} ; retreat
  ; Step 3306, bar 1468
  LIN {X 13535.893,Y 2029.899,Z 855.478,A -89.96659,B 0.00000,C -180.00000} ; outside
  LIN {X 13535.893,Y 2029.899,Z -132.531,A -89.96659,B 0.00000,C -180.00000} ; preinsert
  LIN {X 13535.893,Y 2029.899,Z -382.531,A -89.96659,B 0.00000,C -180.00000} ; insert
  LIN {X 13535.893,Y 2029.899,Z -382.531,A -89.96659,B 0.00000,C -180.00000} ; release
  LIN {X 13535.893,Y 2029.899,Z -82.531,A -89.96659,B 0.00000,C -180.00000} ; retreat
  ; Step 3307, bar 1470
  LIN {X 13635.893,Y 2029.899,Z 855.478,A -89.96659,B 0.00000,C -180.00000} ; outside
  LIN {X 13635.893,Y 2029.899,Z -132.531,A -89.96659,B 0.00000,C -180.00000} ; preinsert
  LIN {X 13635.893,Y 2029.899,Z -382.531,A -89.96659,B 0.00000,C -180.00000} ; insert
  LIN {X 13635.893,Y 2029.899,Z -382.531,A -89.96659,B 0.00000,C -180.00000} ; release
  LIN {X 13635.893,Y 2029.899,Z -82.531,A -89.96659,B 0.00000,C -180.00000} ; retreat
  ; Step 3308, bar 1472
  LIN {X 13735.893,Y 2029.899,Z 855.478,A -89.96659,B 0.00000,C -180.00000} ; outside
  LIN {X 13735.893,Y 2029.899,Z -132.531,A -89.96659,B 0.00000,C -180.00000} ; preinsert
  LIN {X 13735.893,Y 2029.899,Z -382.531,A -89.96659,B 0.00000,C -180.00000} ; insert
  LIN {X 13735.893,Y 2029.899,Z -382.531,A -89.96659,B 0.00000,C -180.00000} ; release
  LIN {X 13735.893,Y 2029.899,Z -82.531,A -89.96659,B 0.00000,C -180.00000} ; retreat
  ; Step 3309, bar 1474
  LIN {X 13835.893,Y 2029.899,Z 855.478,A -89.96659,B 0.00000,C -180.00000} ; outside
  LIN {X 13835.893,Y 2029.899,Z -132.531,A -89.96659,B 0.00000,C -180.00000} ; preinsert
  LIN {X 13835.893,Y 2029.899,Z -382.531,A -89.96659,B 0.00000,C -180.00000} ; insert
  LIN {X 13835.893,Y 2029.899,Z -382.531,A -89.96659,B 0.00000,C -180.00000} ; release
  LIN {X 13835.893,Y 2029.899,Z -82.531,A -89.96659,B 0.00000,C -180.00000} ; retreat
  ; Step 3310, bar 1476
  LIN {X 14135.893,Y 2029.899,Z 855.478,A -89.96659,B 0.00000,C -180.00000} ; outside
  LIN {X 14135.893,Y 2029.899,Z -132.531,A -89.96659,B 0.00000,C -180.00000} ; preinsert
  LIN {X 14135.893,Y 2029.899,Z -382.531,A -89.96659,B 0.00000,C -180.00000} ; insert
  LIN {X 14135.893,Y 2029.899,Z -382.531,A -89.96659,B 0.00000,C -180.00000} ; release
  LIN {X 14135.893,Y 2029.899,Z -82.531,A -89.96659,B 0.00000,C -180.00000} ; retreat
  ; Step 3311, bar 1478
  LIN {X 14235.893,Y 2029.899,Z 855.478,A -89.96659,B 0.00000,C -180.00000} ; outside
  LIN {X 14235.893,Y 2029.899,Z -132.531,A -89.96659,B 0.00000,C -180.00000} ; preinsert
  LIN {X 14235.893,Y 2029.899,Z -382.531,A -89.96659,B 0.00000,C -180.00000} ; insert
  LIN {X 14235.893,Y 2029.899,Z -382.531,A -89.96659,B 0.00000,C -180.00000} ; release
  LIN {X 14235.893,Y 2029.899,Z -82.531,A -89.96659,B 0.00000,C -180.00000} ; retreat
  ; Step 3312, bar 1559
  LIN {X -110.893,Y -2029.899,Z 855.478,A 90.03341,B 0.00000,C 180.00000} ; outside
  LIN {X -110.893,Y -2029.899,Z -132.531,A 90.03341,B 0.00000,C 180.00000} ; preinsert
  LIN {X -110.893,Y -2029.899,Z -382.531,A 90.03341,B 0.00000,C 180.00000} ; insert
  LIN {X -110.893,Y -2029.899,Z -382.531,A 90.03341,B 0.00000,C 180.00000} ; release
  LIN {X -110.893,Y -2029.899,Z -82.531,A 90.03341,B 0.00000,C 180.00000} ; retreat
  ; Step 3313, bar 1561
  LIN {X -235.893,Y -2029.899,Z 855.478,A 90.03341,B 0.00000,C 180.00000} ; outside
  LIN {X -235.893,Y -2029.899,Z -132.531,A 90.03341,B 0.00000,C 180.00000} ; preinsert
  LIN {X -235.893,Y -2029.899,Z -382.531,A 90.03341,B 0.00000,C 180.00000} ; insert
  LIN {X -235.893,Y -2029.899,Z -382.531,A 90.03341,B 0.00000,C 180.00000} ; release
  LIN {X -235.893,Y -2029.899,Z -82.531,A 90.03341,B 0.00000,C 180.00000} ; retreat
  ; Step 3314, bar 1563
  LIN {X -360.893,Y -2029.899,Z 855.478,A 90.03341,B 0.00000,C 180.00000} ; outside
  LIN {X -360.893,Y -2029.899,Z -132.531,A 90.03341,B 0.00000,C 180.00000} ; preinsert
  LIN {X -360.893,Y -2029.899,Z -382.531,A 90.03341,B 0.00000,C 180.00000} ; insert
  LIN {X -360.893,Y -2029.899,Z -382.531,A 90.03341,B 0.00000,C 180.00000} ; release
  LIN {X -360.893,Y -2029.899,Z -82.531,A 90.03341,B 0.00000,C 180.00000} ; retreat
  ; Step 3315, bar 1565
  LIN {X -485.893,Y -2029.899,Z 855.478,A 90.03341,B 0.00000,C 180.00000} ; outside
  LIN {X -485.893,Y -2029.899,Z -132.531,A 90.03341,B 0.00000,C 180.00000} ; preinsert
  LIN {X -485.893,Y -2029.899,Z -382.531,A 90.03341,B 0.00000,C 180.00000} ; insert
  LIN {X -485.893,Y -2029.899,Z -382.531,A 90.03341,B 0.00000,C 180.00000} ; release
  LIN {X -485.893,Y -2029.899,Z -82.531,A 90.03341,B 0.00000,C 180.00000} ; retreat
  ; Step 3316, bar 1567
  LIN {X -610.893,Y -2029.899,Z 855.478,A 90.03341,B 0.00000,C 180.00000} ; outside
  LIN {X -610.893,Y -2029.899,Z -132.531,A 90.03341,B 0.00000,C 180.00000} ; preinsert
  LIN {X -610.893,Y -2029.899,Z -382.531,A 90.03341,B 0.00000,C 180.00000} ; insert
  LIN {X -610.893,Y -2029.899,Z -382.531,A 90.03341,B 0.00000,C 180.00000} ; release
  LIN {X -610.893,Y -2029.899,Z -82.531,A 90.03341,B 0.00000,C 180.00000} ; retreat
  ; Step 3317, bar 1569
  LIN {X -735.893,Y -2029.899,Z 855.478,A 90.03341,B 0.00000,C 180.00000} ; outside
  LIN {X -735.893,Y -2029.899,Z -132.531,A 90.03341,B 0.00000,C 180.00000} ; preinsert
  LIN {X -735.893,Y -2029.899,Z -382.531,A 90.03341,B 0.00000,C 180.00000} ; insert
  LIN {X -735.893,Y -2029.899,Z -382.531,A 90.03341,B 0.00000,C 180.00000} ; release
  LIN {X -735.893,Y -2029.899,Z -82.531,A 90.03341,B 0.00000,C 180.00000} ; retreat
  ; Step 3318, bar 1571
  LIN {X -860.893,Y -2029.899,Z 855.478,A 90.03341,B 0.00000,C 180.00000} ; outside
  LIN {X -860.893,Y -2029.899,Z -132.531,A 90.03341,B 0.00000,C 180.00000} ; preinsert
  LIN {X -860.893,Y -2029.899,Z -382.531,A 90.03341,B 0.00000,C 180.00000} ; insert
  LIN {X -860.893,Y -2029.899,Z -382.531,A 90.03341,B 0.00000,C 180.00000} ; release
  LIN {X -860.893,Y -2029.899,Z -82.531,A 90.03341,B 0.00000,C 180.00000} ; retreat
  ; Step 3319, bar 1573
  LIN {X -985.893,Y -2029.899,Z 855.478,A 90.03341,B 0.00000,C 180.00000} ; outside
  LIN {X -985.893,Y -2029.899,Z -132.531,A 90.03341,B 0.00000,C 180.00000} ; preinsert
  LIN {X -985.893,Y -2029.899,Z -382.531,A 90.03341,B 0.00000,C 180.00000} ; insert
  LIN {X -985.893,Y -2029.899,Z -382.531,A 90.03341,B 0.00000,C 180.00000} ; release
  LIN {X -985.893,Y -2029.899,Z -82.531,A 90.03341,B 0.00000,C 180.00000} ; retreat
  ; Step 3320, bar 1575
  LIN {X -1110.893,Y -2029.899,Z 855.478,A 90.03341,B 0.00000,C 180.00000} ; outside
  LIN {X -1110.893,Y -2029.899,Z -132.531,A 90.03341,B 0.00000,C 180.00000} ; preinsert
  LIN {X -1110.893,Y -2029.899,Z -382.531,A 90.03341,B 0.00000,C 180.00000} ; insert
  LIN {X -1110.893,Y -2029.899,Z -382.531,A 90.03341,B 0.00000,C 180.00000} ; release
  LIN {X -1110.893,Y -2029.899,Z -82.531,A 90.03341,B 0.00000,C 180.00000} ; retreat
  ; Step 3321, bar 1577
  LIN {X -1235.893,Y -2029.899,Z 855.478,A 90.03341,B 0.00000,C 180.00000} ; outside
  LIN {X -1235.893,Y -2029.899,Z -132.531,A 90.03341,B 0.00000,C 180.00000} ; preinsert
  LIN {X -1235.893,Y -2029.899,Z -382.531,A 90.03341,B 0.00000,C 180.00000} ; insert
  LIN {X -1235.893,Y -2029.899,Z -382.531,A 90.03341,B 0.00000,C 180.00000} ; release
  LIN {X -1235.893,Y -2029.899,Z -82.531,A 90.03341,B 0.00000,C 180.00000} ; retreat
  ; Step 3322, bar 1579
  LIN {X -1360.893,Y -2029.899,Z 855.478,A 90.03341,B 0.00000,C 180.00000} ; outside
  LIN {X -1360.893,Y -2029.899,Z -132.531,A 90.03341,B 0.00000,C 180.00000} ; preinsert
  LIN {X -1360.893,Y -2029.899,Z -382.531,A 90.03341,B 0.00000,C 180.00000} ; insert
  LIN {X -1360.893,Y -2029.899,Z -382.531,A 90.03341,B 0.00000,C 180.00000} ; release
  LIN {X -1360.893,Y -2029.899,Z -82.531,A 90.03341,B 0.00000,C 180.00000} ; retreat
  ; Step 3323, bar 1581
  LIN {X -1485.893,Y -2029.899,Z 855.478,A 90.03341,B 0.00000,C 180.00000} ; outside
  LIN {X -1485.893,Y -2029.899,Z -132.531,A 90.03341,B 0.00000,C 180.00000} ; preinsert
  LIN {X -1485.893,Y -2029.899,Z -382.531,A 90.03341,B 0.00000,C 180.00000} ; insert
  LIN {X -1485.893,Y -2029.899,Z -382.531,A 90.03341,B 0.00000,C 180.00000} ; release
  LIN {X -1485.893,Y -2029.899,Z -82.531,A 90.03341,B 0.00000,C 180.00000} ; retreat
  ; Step 3324, bar 1583
  LIN {X -1610.893,Y -2029.899,Z 855.478,A 90.03341,B 0.00000,C 180.00000} ; outside
  LIN {X -1610.893,Y -2029.899,Z -132.531,A 90.03341,B 0.00000,C 180.00000} ; preinsert
  LIN {X -1610.893,Y -2029.899,Z -382.531,A 90.03341,B 0.00000,C 180.00000} ; insert
  LIN {X -1610.893,Y -2029.899,Z -382.531,A 90.03341,B 0.00000,C 180.00000} ; release
  LIN {X -1610.893,Y -2029.899,Z -82.531,A 90.03341,B 0.00000,C 180.00000} ; retreat
  ; Step 3325, bar 1585
  LIN {X -1735.893,Y -2029.899,Z 855.478,A 90.03341,B 0.00000,C 180.00000} ; outside
  LIN {X -1735.893,Y -2029.899,Z -132.531,A 90.03341,B 0.00000,C 180.00000} ; preinsert
  LIN {X -1735.893,Y -2029.899,Z -382.531,A 90.03341,B 0.00000,C 180.00000} ; insert
  LIN {X -1735.893,Y -2029.899,Z -382.531,A 90.03341,B 0.00000,C 180.00000} ; release
  LIN {X -1735.893,Y -2029.899,Z -82.531,A 90.03341,B 0.00000,C 180.00000} ; retreat
  ; Step 3326, bar 1587
  LIN {X -1860.893,Y -2029.899,Z 855.478,A 90.03341,B 0.00000,C 180.00000} ; outside
  LIN {X -1860.893,Y -2029.899,Z -132.531,A 90.03341,B 0.00000,C 180.00000} ; preinsert
  LIN {X -1860.893,Y -2029.899,Z -382.531,A 90.03341,B 0.00000,C 180.00000} ; insert
  LIN {X -1860.893,Y -2029.899,Z -382.531,A 90.03341,B 0.00000,C 180.00000} ; release
  LIN {X -1860.893,Y -2029.899,Z -82.531,A 90.03341,B 0.00000,C 180.00000} ; retreat
  ; Step 3327, bar 1589
  LIN {X -2110.893,Y -2029.899,Z 855.478,A 90.03341,B 0.00000,C 180.00000} ; outside
  LIN {X -2110.893,Y -2029.899,Z -132.531,A 90.03341,B 0.00000,C 180.00000} ; preinsert
  LIN {X -2110.893,Y -2029.899,Z -382.531,A 90.03341,B 0.00000,C 180.00000} ; insert
  LIN {X -2110.893,Y -2029.899,Z -382.531,A 90.03341,B 0.00000,C 180.00000} ; release
  LIN {X -2110.893,Y -2029.899,Z -82.531,A 90.03341,B 0.00000,C 180.00000} ; retreat
  ; Step 3328, bar 1591
  LIN {X -2235.893,Y -2029.899,Z 855.478,A 90.03341,B 0.00000,C 180.00000} ; outside
  LIN {X -2235.893,Y -2029.899,Z -132.531,A 90.03341,B 0.00000,C 180.00000} ; preinsert
  LIN {X -2235.893,Y -2029.899,Z -382.531,A 90.03341,B 0.00000,C 180.00000} ; insert
  LIN {X -2235.893,Y -2029.899,Z -382.531,A 90.03341,B 0.00000,C 180.00000} ; release
  LIN {X -2235.893,Y -2029.899,Z -82.531,A 90.03341,B 0.00000,C 180.00000} ; retreat
  ; Step 3329, bar 1593
  LIN {X -2360.893,Y -2029.899,Z 855.478,A 90.03341,B 0.00000,C 180.00000} ; outside
  LIN {X -2360.893,Y -2029.899,Z -132.531,A 90.03341,B 0.00000,C 180.00000} ; preinsert
  LIN {X -2360.893,Y -2029.899,Z -382.531,A 90.03341,B 0.00000,C 180.00000} ; insert
  LIN {X -2360.893,Y -2029.899,Z -382.531,A 90.03341,B 0.00000,C 180.00000} ; release
  LIN {X -2360.893,Y -2029.899,Z -82.531,A 90.03341,B 0.00000,C 180.00000} ; retreat
  ; Step 3330, bar 1595
  LIN {X -2485.893,Y -2029.899,Z 855.478,A 90.03341,B 0.00000,C 180.00000} ; outside
  LIN {X -2485.893,Y -2029.899,Z -132.531,A 90.03341,B 0.00000,C 180.00000} ; preinsert
  LIN {X -2485.893,Y -2029.899,Z -382.531,A 90.03341,B 0.00000,C 180.00000} ; insert
  LIN {X -2485.893,Y -2029.899,Z -382.531,A 90.03341,B 0.00000,C 180.00000} ; release
  LIN {X -2485.893,Y -2029.899,Z -82.531,A 90.03341,B 0.00000,C 180.00000} ; retreat
  ; Step 3331, bar 1597
  LIN {X -2610.893,Y -2029.899,Z 855.478,A 90.03341,B 0.00000,C 180.00000} ; outside
  LIN {X -2610.893,Y -2029.899,Z -132.531,A 90.03341,B 0.00000,C 180.00000} ; preinsert
  LIN {X -2610.893,Y -2029.899,Z -382.531,A 90.03341,B 0.00000,C 180.00000} ; insert
  LIN {X -2610.893,Y -2029.899,Z -382.531,A 90.03341,B 0.00000,C 180.00000} ; release
  LIN {X -2610.893,Y -2029.899,Z -82.531,A 90.03341,B 0.00000,C 180.00000} ; retreat
  ; Step 3332, bar 1599
  LIN {X -2735.893,Y -2029.899,Z 855.478,A 90.03341,B 0.00000,C 180.00000} ; outside
  LIN {X -2735.893,Y -2029.899,Z -132.531,A 90.03341,B 0.00000,C 180.00000} ; preinsert
  LIN {X -2735.893,Y -2029.899,Z -382.531,A 90.03341,B 0.00000,C 180.00000} ; insert
  LIN {X -2735.893,Y -2029.899,Z -382.531,A 90.03341,B 0.00000,C 180.00000} ; release
  LIN {X -2735.893,Y -2029.899,Z -82.531,A 90.03341,B 0.00000,C 180.00000} ; retreat
  ; Step 3333, bar 1601
  LIN {X -2860.893,Y -2029.899,Z 855.478,A 90.03341,B 0.00000,C 180.00000} ; outside
  LIN {X -2860.893,Y -2029.899,Z -132.531,A 90.03341,B 0.00000,C 180.00000} ; preinsert
  LIN {X -2860.893,Y -2029.899,Z -382.531,A 90.03341,B 0.00000,C 180.00000} ; insert
  LIN {X -2860.893,Y -2029.899,Z -382.531,A 90.03341,B 0.00000,C 180.00000} ; release
  LIN {X -2860.893,Y -2029.899,Z -82.531,A 90.03341,B 0.00000,C 180.00000} ; retreat
  ; Step 3334, bar 1603
  LIN {X -2985.893,Y -2029.899,Z 855.478,A 90.03341,B 0.00000,C 180.00000} ; outside
  LIN {X -2985.893,Y -2029.899,Z -132.531,A 90.03341,B 0.00000,C 180.00000} ; preinsert
  LIN {X -2985.893,Y -2029.899,Z -382.531,A 90.03341,B 0.00000,C 180.00000} ; insert
  LIN {X -2985.893,Y -2029.899,Z -382.531,A 90.03341,B 0.00000,C 180.00000} ; release
  LIN {X -2985.893,Y -2029.899,Z -82.531,A 90.03341,B 0.00000,C 180.00000} ; retreat
  ; Step 3335, bar 1605
  LIN {X -3110.893,Y -2029.899,Z 855.478,A 90.03341,B 0.00000,C 180.00000} ; outside
  LIN {X -3110.893,Y -2029.899,Z -132.531,A 90.03341,B 0.00000,C 180.00000} ; preinsert
  LIN {X -3110.893,Y -2029.899,Z -382.531,A 90.03341,B 0.00000,C 180.00000} ; insert
  LIN {X -3110.893,Y -2029.899,Z -382.531,A 90.03341,B 0.00000,C 180.00000} ; release
  LIN {X -3110.893,Y -2029.899,Z -82.531,A 90.03341,B 0.00000,C 180.00000} ; retreat
  ; Step 3336, bar 1607
  LIN {X -3235.893,Y -2029.899,Z 855.478,A 90.03341,B 0.00000,C 180.00000} ; outside
  LIN {X -3235.893,Y -2029.899,Z -132.531,A 90.03341,B 0.00000,C 180.00000} ; preinsert
  LIN {X -3235.893,Y -2029.899,Z -382.531,A 90.03341,B 0.00000,C 180.00000} ; insert
  LIN {X -3235.893,Y -2029.899,Z -382.531,A 90.03341,B 0.00000,C 180.00000} ; release
  LIN {X -3235.893,Y -2029.899,Z -82.531,A 90.03341,B 0.00000,C 180.00000} ; retreat
  ; Step 3337, bar 1609
  LIN {X -3360.893,Y -2029.899,Z 855.478,A 90.03341,B 0.00000,C 180.00000} ; outside
  LIN {X -3360.893,Y -2029.899,Z -132.531,A 90.03341,B 0.00000,C 180.00000} ; preinsert
  LIN {X -3360.893,Y -2029.899,Z -382.531,A 90.03341,B 0.00000,C 180.00000} ; insert
  LIN {X -3360.893,Y -2029.899,Z -382.531,A 90.03341,B 0.00000,C 180.00000} ; release
  LIN {X -3360.893,Y -2029.899,Z -82.531,A 90.03341,B 0.00000,C 180.00000} ; retreat
  ; Step 3338, bar 1611
  LIN {X -3485.893,Y -2029.899,Z 855.478,A 90.03341,B 0.00000,C 180.00000} ; outside
  LIN {X -3485.893,Y -2029.899,Z -132.531,A 90.03341,B 0.00000,C 180.00000} ; preinsert
  LIN {X -3485.893,Y -2029.899,Z -382.531,A 90.03341,B 0.00000,C 180.00000} ; insert
  LIN {X -3485.893,Y -2029.899,Z -382.531,A 90.03341,B 0.00000,C 180.00000} ; release
  LIN {X -3485.893,Y -2029.899,Z -82.531,A 90.03341,B 0.00000,C 180.00000} ; retreat
  ; Step 3339, bar 1613
  LIN {X -3610.893,Y -2029.899,Z 855.478,A 90.03341,B 0.00000,C 180.00000} ; outside
  LIN {X -3610.893,Y -2029.899,Z -132.531,A 90.03341,B 0.00000,C 180.00000} ; preinsert
  LIN {X -3610.893,Y -2029.899,Z -382.531,A 90.03341,B 0.00000,C 180.00000} ; insert
  LIN {X -3610.893,Y -2029.899,Z -382.531,A 90.03341,B 0.00000,C 180.00000} ; release
  LIN {X -3610.893,Y -2029.899,Z -82.531,A 90.03341,B 0.00000,C 180.00000} ; retreat
  ; Step 3340, bar 1615
  LIN {X -3735.893,Y -2029.899,Z 855.478,A 90.03341,B 0.00000,C 180.00000} ; outside
  LIN {X -3735.893,Y -2029.899,Z -132.531,A 90.03341,B 0.00000,C 180.00000} ; preinsert
  LIN {X -3735.893,Y -2029.899,Z -382.531,A 90.03341,B 0.00000,C 180.00000} ; insert
  LIN {X -3735.893,Y -2029.899,Z -382.531,A 90.03341,B 0.00000,C 180.00000} ; release
  LIN {X -3735.893,Y -2029.899,Z -82.531,A 90.03341,B 0.00000,C 180.00000} ; retreat
  ; Step 3341, bar 1617
  LIN {X -3860.893,Y -2029.899,Z 855.478,A 90.03341,B 0.00000,C 180.00000} ; outside
  LIN {X -3860.893,Y -2029.899,Z -132.531,A 90.03341,B 0.00000,C 180.00000} ; preinsert
  LIN {X -3860.893,Y -2029.899,Z -382.531,A 90.03341,B 0.00000,C 180.00000} ; insert
  LIN {X -3860.893,Y -2029.899,Z -382.531,A 90.03341,B 0.00000,C 180.00000} ; release
  LIN {X -3860.893,Y -2029.899,Z -82.531,A 90.03341,B 0.00000,C 180.00000} ; retreat
  ; Step 3342, bar 1619
  LIN {X -3985.893,Y -2029.899,Z 855.478,A 90.03341,B 0.00000,C 180.00000} ; outside
  LIN {X -3985.893,Y -2029.899,Z -132.531,A 90.03341,B 0.00000,C 180.00000} ; preinsert
  LIN {X -3985.893,Y -2029.899,Z -382.531,A 90.03341,B 0.00000,C 180.00000} ; insert
  LIN {X -3985.893,Y -2029.899,Z -382.531,A 90.03341,B 0.00000,C 180.00000} ; release
  LIN {X -3985.893,Y -2029.899,Z -82.531,A 90.03341,B 0.00000,C 180.00000} ; retreat
  ; Step 3343, bar 1621
  LIN {X -4110.893,Y -2029.899,Z 855.478,A 90.03341,B 0.00000,C 180.00000} ; outside
  LIN {X -4110.893,Y -2029.899,Z -132.531,A 90.03341,B 0.00000,C 180.00000} ; preinsert
  LIN {X -4110.893,Y -2029.899,Z -382.531,A 90.03341,B 0.00000,C 180.00000} ; insert
  LIN {X -4110.893,Y -2029.899,Z -382.531,A 90.03341,B 0.00000,C 180.00000} ; release
  LIN {X -4110.893,Y -2029.899,Z -82.531,A 90.03341,B 0.00000,C 180.00000} ; retreat
  ; Step 3344, bar 1623
  LIN {X -4235.893,Y -2029.899,Z 855.478,A 90.03341,B 0.00000,C 180.00000} ; outside
  LIN {X -4235.893,Y -2029.899,Z -132.531,A 90.03341,B 0.00000,C 180.00000} ; preinsert
  LIN {X -4235.893,Y -2029.899,Z -382.531,A 90.03341,B 0.00000,C 180.00000} ; insert
  LIN {X -4235.893,Y -2029.899,Z -382.531,A 90.03341,B 0.00000,C 180.00000} ; release
  LIN {X -4235.893,Y -2029.899,Z -82.531,A 90.03341,B 0.00000,C 180.00000} ; retreat
  ; Step 3345, bar 1625
  LIN {X -4360.893,Y -2029.899,Z 855.478,A 90.03341,B 0.00000,C 180.00000} ; outside
  LIN {X -4360.893,Y -2029.899,Z -132.531,A 90.03341,B 0.00000,C 180.00000} ; preinsert
  LIN {X -4360.893,Y -2029.899,Z -382.531,A 90.03341,B 0.00000,C 180.00000} ; insert
  LIN {X -4360.893,Y -2029.899,Z -382.531,A 90.03341,B 0.00000,C 180.00000} ; release
  LIN {X -4360.893,Y -2029.899,Z -82.531,A 90.03341,B 0.00000,C 180.00000} ; retreat
  ; Step 3346, bar 1627
  LIN {X -4485.893,Y -2029.899,Z 855.478,A 90.03341,B 0.00000,C 180.00000} ; outside
  LIN {X -4485.893,Y -2029.899,Z -132.531,A 90.03341,B 0.00000,C 180.00000} ; preinsert
  LIN {X -4485.893,Y -2029.899,Z -382.531,A 90.03341,B 0.00000,C 180.00000} ; insert
  LIN {X -4485.893,Y -2029.899,Z -382.531,A 90.03341,B 0.00000,C 180.00000} ; release
  LIN {X -4485.893,Y -2029.899,Z -82.531,A 90.03341,B 0.00000,C 180.00000} ; retreat
  ; Step 3347, bar 1629
  LIN {X -4610.893,Y -2029.899,Z 855.478,A 90.03341,B 0.00000,C 180.00000} ; outside
  LIN {X -4610.893,Y -2029.899,Z -132.531,A 90.03341,B 0.00000,C 180.00000} ; preinsert
  LIN {X -4610.893,Y -2029.899,Z -382.531,A 90.03341,B 0.00000,C 180.00000} ; insert
  LIN {X -4610.893,Y -2029.899,Z -382.531,A 90.03341,B 0.00000,C 180.00000} ; release
  LIN {X -4610.893,Y -2029.899,Z -82.531,A 90.03341,B 0.00000,C 180.00000} ; retreat
  ; Step 3348, bar 1631
  LIN {X -4735.893,Y -2029.899,Z 855.478,A 90.03341,B 0.00000,C 180.00000} ; outside
  LIN {X -4735.893,Y -2029.899,Z -132.531,A 90.03341,B 0.00000,C 180.00000} ; preinsert
  LIN {X -4735.893,Y -2029.899,Z -382.531,A 90.03341,B 0.00000,C 180.00000} ; insert
  LIN {X -4735.893,Y -2029.899,Z -382.531,A 90.03341,B 0.00000,C 180.00000} ; release
  LIN {X -4735.893,Y -2029.899,Z -82.531,A 90.03341,B 0.00000,C 180.00000} ; retreat
  ; Step 3349, bar 1633
  LIN {X -4860.893,Y -2029.899,Z 855.478,A 90.03341,B 0.00000,C 180.00000} ; outside
  LIN {X -4860.893,Y -2029.899,Z -132.531,A 90.03341,B 0.00000,C 180.00000} ; preinsert
  LIN {X -4860.893,Y -2029.899,Z -382.531,A 90.03341,B 0.00000,C 180.00000} ; insert
  LIN {X -4860.893,Y -2029.899,Z -382.531,A 90.03341,B 0.00000,C 180.00000} ; release
